LIN {X 0,Y 524.001,Z 123.213,A -85,B 0,C 180,E1 -4868.484,E2 -4868.484} C_VEL
LIN {X 0,Y 524.001,Z 123.208,A -85,B 0,C 180,E1 -4871.74,E2 -4871.74} C_VEL
LIN {X 0,Y 523.991,Z 123.214,A -85,B 0,C 180,E1 -4875.052,E2 -4875.052} C_VEL
LIN {X 0,Y 523.962,Z 123.215,A -85,B 0,C 180,E1 -4877.969,E2 -4877.969} C_VEL
LIN {X 0,Y 523.97,Z 123.219,A -85,B 0,C 180,E1 -4880.41,E2 -4880.41} C_VEL
LIN {X 0,Y 523.909,Z 123.226,A -85,B 0,C 180,E1 -4882.893,E2 -4882.893} C_VEL
LIN {X 0,Y 523.95,Z 123.217,A -85,B 0,C 180,E1 -4885.419,E2 -4885.419} C_VEL
LIN {X 0,Y 523.968,Z 123.218,A -85,B 0,C 180,E1 -4887.999,E2 -4887.999} C_VEL
LIN {X 0,Y 523.945,Z 123.22,A -85,B 0,C 180,E1 -4890.855,E2 -4890.855} C_VEL
LIN {X 0,Y 523.961,Z 123.218,A -85,B 0,C 180,E1 -4893.735,E2 -4893.735} C_VEL
LIN {X 0,Y 524.017,Z 123.347,A -85,B 0,C 180,E1 -4894.881,E2 -4894.881} C_VEL
LIN {X 0,Y 524.386,Z 128.549,A -85,B 0,C 180,E1 -4895.898,E2 -4895.898} C_VEL
LIN {X 0,Y 524.291,Z 138.967,A -85,B 0,C 180,E1 -4897.913,E2 -4897.913} C_VEL
LIN {X 0,Y 525.934,Z 147.356,A -85,B 0,C 180,E1 -4898.081,E2 -4898.081} C_VEL
LIN {X 0,Y 525.786,Z 195.44,A -85,B 0,C 180,E1 -4898.751,E2 -4898.751} C_VEL
LIN {X 0,Y 525.168,Z 201.285,A -85,B 0,C 180,E1 -4898.816,E2 -4898.816} C_VEL
LIN {X 0,Y 519.401,Z 220.267,A -85,B 0,C 180,E1 -4898.921,E2 -4898.921} C_VEL
LIN {X 0,Y 518.753,Z 226.114,A -85,B 0,C 180,E1 -4898.986,E2 -4898.986} C_VEL
LIN {X 0,Y 518.635,Z 247.138,A -85,B 0,C 180,E1 -4899.309,E2 -4899.309} C_VEL
LIN {X 0,Y 518.446,Z 260.421,A -85,B 0,C 180,E1 -4899.672,E2 -4899.672} C_VEL
LIN {X 0,Y 518.242,Z 272.646,A -85,B 0,C 180,E1 -4900.166,E2 -4900.166} C_VEL
LIN {X 0,Y 517.974,Z 284.77,A -85,B 0,C 180,E1 -4900.83,E2 -4900.83} C_VEL
LIN {X 0,Y 517.696,Z 296.092,A -85,B 0,C 180,E1 -4901.626,E2 -4901.626} C_VEL
LIN {X 0,Y 517.426,Z 306.152,A -85,B 0,C 180,E1 -4902.511,E2 -4902.511} C_VEL
LIN {X 0,Y 517.15,Z 314.732,A -85,B 0,C 180,E1 -4903.435,E2 -4903.435} C_VEL
LIN {X 0,Y 516.882,Z 322.531,A -85,B 0,C 180,E1 -4904.452,E2 -4904.452} C_VEL
LIN {X 0,Y 516.675,Z 329.356,A -85,B 0,C 180,E1 -4905.536,E2 -4905.536} C_VEL
LIN {X 0,Y 516.508,Z 336.123,A -85,B 0,C 180,E1 -4906.882,E2 -4906.882} C_VEL
LIN {X 0,Y 516.419,Z 341.098,A -85,B 0,C 180,E1 -4908.176,E2 -4908.176} C_VEL
LIN {X 0,Y 516.322,Z 345.19,A -85,B 0,C 180,E1 -4909.663,E2 -4909.663} C_VEL
LIN {X 0,Y 516.228,Z 347.859,A -85,B 0,C 180,E1 -4911.226,E2 -4911.226} C_VEL
LIN {X 0,Y 516.202,Z 348.684,A -85,B 0,C 180,E1 -4912.218,E2 -4912.218} C_VEL
LIN {X 0,Y 516.215,Z 348.842,A -85,B 0,C 180,E1 -4913.442,E2 -4913.442} C_VEL
LIN {X 0,Y 516.204,Z 347.924,A -85,B 0,C 180,E1 -4914.774,E2 -4914.774} C_VEL
LIN {X 0,Y 516.335,Z 345.799,A -85,B 0,C 180,E1 -4916.128,E2 -4916.128} C_VEL
LIN {X 0,Y 516.364,Z 342.184,A -85,B 0,C 180,E1 -4917.549,E2 -4917.549} C_VEL
LIN {X 0,Y 516.476,Z 337.486,A -85,B 0,C 180,E1 -4918.863,E2 -4918.863} C_VEL
LIN {X 0,Y 516.65,Z 331.294,A -85,B 0,C 180,E1 -4920.186,E2 -4920.186} C_VEL
LIN {X 0,Y 516.858,Z 324.311,A -85,B 0,C 180,E1 -4921.36,E2 -4921.36} C_VEL
LIN {X 0,Y 517.048,Z 316.091,A -85,B 0,C 180,E1 -4922.475,E2 -4922.475} C_VEL
LIN {X 0,Y 517.361,Z 307.081,A -85,B 0,C 180,E1 -4923.47,E2 -4923.47} C_VEL
LIN {X 0,Y 517.635,Z 297.279,A -85,B 0,C 180,E1 -4924.357,E2 -4924.357} C_VEL
LIN {X 0,Y 517.885,Z 286.81,A -85,B 0,C 180,E1 -4925.122,E2 -4925.122} C_VEL
LIN {X 0,Y 518.158,Z 274.714,A -85,B 0,C 180,E1 -4925.813,E2 -4925.813} C_VEL
LIN {X 0,Y 518.398,Z 262.998,A -85,B 0,C 180,E1 -4926.32,E2 -4926.32} C_VEL
LIN {X 0,Y 518.596,Z 250.647,A -85,B 0,C 180,E1 -4926.7,E2 -4926.7} C_VEL
LIN {X 0,Y 518.693,Z 236.856,A -85,B 0,C 180,E1 -4926.953,E2 -4926.953} C_VEL
LIN {X 0,Y 519.143,Z 148.357,A -85,B 0,C 180,E1 -4928.196,E2 -4928.196} C_VEL
LIN {X 0,Y 517.213,Z 138.968,A -85,B 0,C 180,E1 -4928.398,E2 -4928.398} C_VEL
LIN {X 0,Y 517.29,Z 127.147,A -85,B 0,C 180,E1 -4930.764,E2 -4930.764} C_VEL
LIN {X 0,Y 516.945,Z 124.095,A -85,B 0,C 180,E1 -4931.42,E2 -4931.42} C_VEL
LIN {X 0,Y 516.945,Z 124.089,A -85,B 0,C 180,E1 -4934.854,E2 -4934.854} C_VEL
LIN {X 0,Y 516.966,Z 124.086,A -85,B 0,C 180,E1 -4938.234,E2 -4938.234} C_VEL
LIN {X 0,Y 516.965,Z 124.091,A -85,B 0,C 180,E1 -4941.4,E2 -4941.4} C_VEL
LIN {X 0,Y 517.003,Z 124.085,A -85,B 0,C 180,E1 -4943.757,E2 -4943.757} C_VEL
LIN {X 0,Y 517.009,Z 124.081,A -85,B 0,C 180,E1 -4946.883,E2 -4946.883} C_VEL
LIN {X 0,Y 517.093,Z 124.075,A -85,B 0,C 180,E1 -4949.221,E2 -4949.221} C_VEL
LIN {X 0,Y 517.084,Z 124.07,A -85,B 0,C 180,E1 -4952.337,E2 -4952.337} C_VEL
LIN {X 0,Y 517.027,Z 124.082,A -85,B 0,C 180,E1 -4955.46,E2 -4955.46} C_VEL
LIN {X 0,Y 516.956,Z 124.088,A -85,B 0,C 180,E1 -4958.601,E2 -4958.601} C_VEL
LIN {X 0,Y 516.952,Z 124.087,A -85,B 0,C 180,E1 -4961.807,E2 -4961.807} C_VEL
LIN {X 0,Y 516.945,Z 124.093,A -85,B 0,C 180,E1 -4965.146,E2 -4965.146} C_VEL
LIN {X 0,Y 516.916,Z 124.092,A -85,B 0,C 180,E1 -4968.222,E2 -4968.222} C_VEL
LIN {X 0,Y 516.912,Z 124.098,A -85,B 0,C 180,E1 -4970.701,E2 -4970.701} C_VEL
LIN {X 0,Y 516.903,Z 124.093,A -85,B 0,C 180,E1 -4974.072,E2 -4974.072} C_VEL
LIN {X 0,Y 516.924,Z 124.099,A -85,B 0,C 180,E1 -4976.658,E2 -4976.658} C_VEL
LIN {X 0,Y 516.909,Z 124.092,A -85,B 0,C 180,E1 -4979.523,E2 -4979.523} C_VEL
LIN {X 0,Y 516.893,Z 124.103,A -85,B 0,C 180,E1 -4982.543,E2 -4982.543} C_VEL
LIN {X 0,Y 516.865,Z 124.097,A -85,B 0,C 180,E1 -4985.329,E2 -4985.329} C_VEL
LIN {X 0,Y 516.88,Z 124.098,A -85,B 0,C 180,E1 -4987.943,E2 -4987.943} C_VEL
LIN {X 0,Y 516.882,Z 124.098,A -85,B 0,C 180,E1 -4990.741,E2 -4990.741} C_VEL
LIN {X 0,Y 516.883,Z 124.097,A -85,B 0,C 180,E1 -4992.831,E2 -4992.831} C_VEL
LIN {X 0,Y 516.921,Z 124.09,A -85,B 0,C 180,E1 -4995.01,E2 -4995.01} C_VEL
LIN {X 0,Y 516.913,Z 124.096,A -85,B 0,C 180,E1 -4998.398,E2 -4998.398} C_VEL
LIN {X 0,Y 516.881,Z 124.095,A -85,B 0,C 180,E1 -5001.284,E2 -5001.284} C_VEL
LIN {X 0,Y 516.885,Z 124.1,A -85,B 0,C 180,E1 -5004.221,E2 -5004.221} C_VEL
LIN {X 0,Y 516.893,Z 124.094,A -85,B 0,C 180,E1 -5007.053,E2 -5007.053} C_VEL
LIN {X 0,Y 516.899,Z 124.101,A -85,B 0,C 180,E1 -5009.797,E2 -5009.797} C_VEL
LIN {X 0,Y 516.924,Z 124.091,A -85,B 0,C 180,E1 -5012.467,E2 -5012.467} C_VEL
LIN {X 0,Y 516.873,Z 124.097,A -85,B 0,C 180,E1 -5015.07,E2 -5015.07} C_VEL
LIN {X 0,Y 516.866,Z 124.105,A -85,B 0,C 180,E1 -5017.622,E2 -5017.622} C_VEL
LIN {X 0,Y 516.93,Z 124.091,A -85,B 0,C 180,E1 -5020.13,E2 -5020.13} C_VEL
LIN {X 0,Y 516.927,Z 124.089,A -85,B 0,C 180,E1 -5022.596,E2 -5022.596} C_VEL
LIN {X 0,Y 516.949,Z 124.089,A -85,B 0,C 180,E1 -5025.03,E2 -5025.03} C_VEL
LIN {X 0,Y 516.964,Z 124.085,A -85,B 0,C 180,E1 -5028.234,E2 -5028.234} C_VEL
LIN {X 0,Y 516.968,Z 124.092,A -85,B 0,C 180,E1 -5031.4,E2 -5031.4} C_VEL
LIN {X 0,Y 517.014,Z 124.081,A -85,B 0,C 180,E1 -5033.757,E2 -5033.757} C_VEL
LIN {X 0,Y 517.084,Z 124.072,A -85,B 0,C 180,E1 -5037.663,E2 -5037.663} C_VEL
LIN {X 0,Y 517.091,Z 124.073,A -85,B 0,C 180,E1 -5040.779,E2 -5040.779} C_VEL
LIN {X 0,Y 517.011,Z 124.086,A -85,B 0,C 180,E1 -5043.117,E2 -5043.117} C_VEL
LIN {X 0,Y 517.002,Z 124.081,A -85,B 0,C 180,E1 -5046.243,E2 -5046.243} C_VEL
LIN {X 0,Y 516.951,Z 124.088,A -85,B 0,C 180,E1 -5049.389,E2 -5049.389} C_VEL
LIN {X 0,Y 516.951,Z 124.086,A -85,B 0,C 180,E1 -5051.807,E2 -5051.807} C_VEL
LIN {X 0,Y 516.943,Z 124.09,A -85,B 0,C 180,E1 -5055.147,E2 -5055.147} C_VEL
LIN {X 0,Y 516.924,Z 124.093,A -85,B 0,C 180,E1 -5058.222,E2 -5058.222} C_VEL
LIN {X 0,Y 516.912,Z 124.098,A -85,B 0,C 180,E1 -5060.702,E2 -5060.702} C_VEL
LIN {X 0,Y 516.903,Z 124.095,A -85,B 0,C 180,E1 -5064.073,E2 -5064.073} C_VEL
LIN {X 0,Y 516.924,Z 124.095,A -85,B 0,C 180,E1 -5066.658,E2 -5066.658} C_VEL
LIN {X 0,Y 516.911,Z 124.092,A -85,B 0,C 180,E1 -5069.524,E2 -5069.524} C_VEL
LIN {X 0,Y 516.895,Z 124.098,A -85,B 0,C 180,E1 -5072.544,E2 -5072.544} C_VEL
LIN {X 0,Y 516.866,Z 124.097,A -85,B 0,C 180,E1 -5075.33,E2 -5075.33} C_VEL
LIN {X 0,Y 516.882,Z 124.101,A -85,B 0,C 180,E1 -5077.944,E2 -5077.944} C_VEL
LIN {X 0,Y 516.905,Z 124.093,A -85,B 0,C 180,E1 -5080.74,E2 -5080.74} C_VEL
LIN {X 0,Y 516.883,Z 124.102,A -85,B 0,C 180,E1 -5083.903,E2 -5083.903} C_VEL
LIN {X 0,Y 516.883,Z 124.101,A -85,B 0,C 180,E1 -5086.107,E2 -5086.107} C_VEL
LIN {X 0,Y 516.906,Z 124.093,A -85,B 0,C 180,E1 -5089.261,E2 -5089.261} C_VEL
LIN {X 0,Y 516.865,Z 124.1,A -85,B 0,C 180,E1 -5092.275,E2 -5092.275} C_VEL
LIN {X 0,Y 516.884,Z 124.096,A -85,B 0,C 180,E1 -5095.176,E2 -5095.176} C_VEL
LIN {X 0,Y 516.875,Z 124.1,A -85,B 0,C 180,E1 -5097.975,E2 -5097.975} C_VEL
LIN {X 0,Y 516.924,Z 124.092,A -85,B 0,C 180,E1 -5100.696,E2 -5100.696} C_VEL
LIN {X 0,Y 516.945,Z 124.096,A -85,B 0,C 180,E1 -5103.804,E2 -5103.804} C_VEL
LIN {X 0,Y 516.98,Z 124.198,A -85,B 0,C 180,E1 -5104.457,E2 -5104.457} C_VEL
LIN {X 0,Y 518.589,Z 132.719,A -85,B 0,C 180,E1 -5105.837,E2 -5105.837} C_VEL
LIN {X 0,Y 518.195,Z 147.747,A -85,B 0,C 180,E1 -5108.101,E2 -5108.101} C_VEL
LIN {X 0,Y 517.814,Z 164.388,A -85,B 0,C 180,E1 -5110.578,E2 -5110.578} C_VEL
LIN {X 0,Y 517.443,Z 183.777,A -85,B 0,C 180,E1 -5113.428,E2 -5113.428} C_VEL
LIN {X 0,Y 517.219,Z 191.987,A -85,B 0,C 180,E1 -5114.624,E2 -5114.624} C_VEL
LIN {X 0,Y 518.995,Z 205.511,A -85,B 0,C 180,E1 -5114.873,E2 -5114.873} C_VEL
LIN {X 0,Y 518.582,Z 300.996,A -85,B 0,C 180,E1 -5116.231,E2 -5116.231} C_VEL
LIN {X 0,Y 518.283,Z 314.183,A -85,B 0,C 180,E1 -5116.572,E2 -5116.572} C_VEL
LIN {X 0,Y 518.026,Z 326.893,A -85,B 0,C 180,E1 -5117.065,E2 -5117.065} C_VEL
LIN {X 0,Y 517.759,Z 338.435,A -85,B 0,C 180,E1 -5117.67,E2 -5117.67} C_VEL
LIN {X 0,Y 517.447,Z 349.9,A -85,B 0,C 180,E1 -5118.443,E2 -5118.443} C_VEL
LIN {X 0,Y 517.156,Z 360.428,A -85,B 0,C 180,E1 -5119.33,E2 -5119.33} C_VEL
LIN {X 0,Y 516.86,Z 369.035,A -85,B 0,C 180,E1 -5120.214,E2 -5120.214} C_VEL
LIN {X 0,Y 516.674,Z 376.981,A -85,B 0,C 180,E1 -5121.198,E2 -5121.198} C_VEL
LIN {X 0,Y 516.515,Z 384.746,A -85,B 0,C 180,E1 -5122.376,E2 -5122.376} C_VEL
LIN {X 0,Y 516.374,Z 391.895,A -85,B 0,C 180,E1 -5123.749,E2 -5123.749} C_VEL
LIN {X 0,Y 516.312,Z 396.653,A -85,B 0,C 180,E1 -5124.924,E2 -5124.924} C_VEL
LIN {X 0,Y 516.37,Z 400.293,A -85,B 0,C 180,E1 -5126.098,E2 -5126.098} C_VEL
LIN {X 0,Y 516.327,Z 402.167,A -85,B 0,C 180,E1 -5126.879,E2 -5126.879} C_VEL
LIN {X 0,Y 516.266,Z 403.569,A -85,B 0,C 180,E1 -5127.659,E2 -5127.659} C_VEL
LIN {X 0,Y 516.182,Z 405.175,A -85,B 0,C 180,E1 -5129.22,E2 -5129.22} C_VEL
LIN {X 0,Y 516.186,Z 405.389,A -85,B 0,C 180,E1 -5130,E2 -5130} C_VEL
LIN {X 0,Y 516.182,Z 405.167,A -85,B 0,C 180,E1 -5130.78,E2 -5130.78} C_VEL
LIN {X 0,Y 516.266,Z 403.546,A -85,B 0,C 180,E1 -5132.341,E2 -5132.341} C_VEL
LIN {X 0,Y 516.327,Z 402.135,A -85,B 0,C 180,E1 -5133.121,E2 -5133.121} C_VEL
LIN {X 0,Y 516.312,Z 399.164,A -85,B 0,C 180,E1 -5134.293,E2 -5134.293} C_VEL
LIN {X 0,Y 516.388,Z 395.149,A -85,B 0,C 180,E1 -5135.467,E2 -5135.467} C_VEL
LIN {X 0,Y 516.427,Z 388.964,A -85,B 0,C 180,E1 -5136.84,E2 -5136.84} C_VEL
LIN {X 0,Y 516.564,Z 382.225,A -85,B 0,C 180,E1 -5138.016,E2 -5138.016} C_VEL
LIN {X 0,Y 516.751,Z 373.857,A -85,B 0,C 180,E1 -5139.195,E2 -5139.195} C_VEL
LIN {X 0,Y 516.952,Z 365.274,A -85,B 0,C 180,E1 -5140.18,E2 -5140.18} C_VEL
LIN {X 0,Y 517.294,Z 354.681,A -85,B 0,C 180,E1 -5141.163,E2 -5141.163} C_VEL
LIN {X 0,Y 517.565,Z 343.007,A -85,B 0,C 180,E1 -5142.033,E2 -5142.033} C_VEL
LIN {X 0,Y 517.91,Z 330.721,A -85,B 0,C 180,E1 -5142.739,E2 -5142.739} C_VEL
LIN {X 0,Y 518.17,Z 318.202,A -85,B 0,C 180,E1 -5143.281,E2 -5143.281} C_VEL
LIN {X 0,Y 518.48,Z 305.218,A -85,B 0,C 180,E1 -5143.672,E2 -5143.672} C_VEL
LIN {X 0,Y 518.647,Z 289.599,A -85,B 0,C 180,E1 -5143.942,E2 -5143.942} C_VEL
LIN {X 0,Y 518.951,Z 204.029,A -85,B 0,C 180,E1 -5145.145,E2 -5145.145} C_VEL
LIN {X 0,Y 517.226,Z 191.497,A -85,B 0,C 180,E1 -5145.39,E2 -5145.39} C_VEL
LIN {X 0,Y 517.649,Z 169.331,A -85,B 0,C 180,E1 -5148.606,E2 -5148.606} C_VEL
LIN {X 0,Y 518.082,Z 149.697,A -85,B 0,C 180,E1 -5151.485,E2 -5151.485} C_VEL
LIN {X 0,Y 518.414,Z 132.799,A -85,B 0,C 180,E1 -5153.998,E2 -5153.998} C_VEL
LIN {X 0,Y 516.945,Z 124.094,A -85,B 0,C 180,E1 -5155.383,E2 -5155.383} C_VEL
LIN {X 0,Y 516.92,Z 124.1,A -85,B 0,C 180,E1 -5158.415,E2 -5158.415} C_VEL
LIN {X 0,Y 516.89,Z 124.096,A -85,B 0,C 180,E1 -5161.109,E2 -5161.109} C_VEL
LIN {X 0,Y 516.909,Z 124.098,A -85,B 0,C 180,E1 -5163.966,E2 -5163.966} C_VEL
LIN {X 0,Y 516.877,Z 124.1,A -85,B 0,C 180,E1 -5166.746,E2 -5166.746} C_VEL
LIN {X 0,Y 516.904,Z 124.097,A -85,B 0,C 180,E1 -5169.719,E2 -5169.719} C_VEL
LIN {X 0,Y 516.919,Z 124.096,A -85,B 0,C 180,E1 -5171.774,E2 -5171.774} C_VEL
LIN {X 0,Y 516.923,Z 124.092,A -85,B 0,C 180,E1 -5175.01,E2 -5175.01} C_VEL
LIN {X 0,Y 516.923,Z 124.094,A -85,B 0,C 180,E1 -5178.397,E2 -5178.397} C_VEL
LIN {X 0,Y 516.886,Z 124.095,A -85,B 0,C 180,E1 -5181.284,E2 -5181.284} C_VEL
LIN {X 0,Y 516.87,Z 124.101,A -85,B 0,C 180,E1 -5184.219,E2 -5184.219} C_VEL
LIN {X 0,Y 516.894,Z 124.093,A -85,B 0,C 180,E1 -5187.053,E2 -5187.053} C_VEL
LIN {X 0,Y 516.891,Z 124.1,A -85,B 0,C 180,E1 -5189.796,E2 -5189.796} C_VEL
LIN {X 0,Y 516.925,Z 124.09,A -85,B 0,C 180,E1 -5192.467,E2 -5192.467} C_VEL
LIN {X 0,Y 516.874,Z 124.097,A -85,B 0,C 180,E1 -5195.07,E2 -5195.07} C_VEL
LIN {X 0,Y 516.867,Z 124.102,A -85,B 0,C 180,E1 -5197.621,E2 -5197.621} C_VEL
LIN {X 0,Y 516.931,Z 124.089,A -85,B 0,C 180,E1 -5200.13,E2 -5200.13} C_VEL
LIN {X 0,Y 516.928,Z 124.089,A -85,B 0,C 180,E1 -5202.596,E2 -5202.596} C_VEL
LIN {X 0,Y 516.949,Z 124.089,A -85,B 0,C 180,E1 -5205.03,E2 -5205.03} C_VEL
LIN {X 0,Y 516.964,Z 124.084,A -85,B 0,C 180,E1 -5208.233,E2 -5208.233} C_VEL
LIN {X 0,Y 516.968,Z 124.09,A -85,B 0,C 180,E1 -5211.399,E2 -5211.399} C_VEL
LIN {X 0,Y 517.014,Z 124.081,A -85,B 0,C 180,E1 -5213.757,E2 -5213.757} C_VEL
LIN {X 0,Y 517.084,Z 124.072,A -85,B 0,C 180,E1 -5217.663,E2 -5217.663} C_VEL
LIN {X 0,Y 517.091,Z 124.073,A -85,B 0,C 180,E1 -5220.779,E2 -5220.779} C_VEL
LIN {X 0,Y 517.011,Z 124.086,A -85,B 0,C 180,E1 -5223.117,E2 -5223.117} C_VEL
LIN {X 0,Y 517.001,Z 124.08,A -85,B 0,C 180,E1 -5226.243,E2 -5226.243} C_VEL
LIN {X 0,Y 516.95,Z 124.089,A -85,B 0,C 180,E1 -5229.389,E2 -5229.389} C_VEL
LIN {X 0,Y 516.95,Z 124.087,A -85,B 0,C 180,E1 -5231.807,E2 -5231.807} C_VEL
LIN {X 0,Y 516.942,Z 124.091,A -85,B 0,C 180,E1 -5235.146,E2 -5235.146} C_VEL
LIN {X 0,Y 516.923,Z 124.094,A -85,B 0,C 180,E1 -5238.222,E2 -5238.222} C_VEL
LIN {X 0,Y 516.91,Z 124.1,A -85,B 0,C 180,E1 -5240.701,E2 -5240.701} C_VEL
LIN {X 0,Y 516.901,Z 124.099,A -85,B 0,C 180,E1 -5244.072,E2 -5244.072} C_VEL
LIN {X 0,Y 516.924,Z 124.099,A -85,B 0,C 180,E1 -5246.658,E2 -5246.658} C_VEL
LIN {X 0,Y 516.909,Z 124.094,A -85,B 0,C 180,E1 -5249.524,E2 -5249.524} C_VEL
LIN {X 0,Y 516.899,Z 124.102,A -85,B 0,C 180,E1 -5252.544,E2 -5252.544} C_VEL
LIN {X 0,Y 517.005,Z 124.223,A -85,B 0,C 180,E1 -5254.757,E2 -5254.757} C_VEL
LIN {X 0,Y 517.418,Z 129.161,A -85,B 0,C 180,E1 -5255.737,E2 -5255.737} C_VEL
LIN {X 0,Y 517.292,Z 139.212,A -85,B 0,C 180,E1 -5257.689,E2 -5257.689} C_VEL
LIN {X 0,Y 519.145,Z 148.956,A -85,B 0,C 180,E1 -5257.898,E2 -5257.898} C_VEL
LIN {X 0,Y 518.753,Z 226.114,A -85,B 0,C 180,E1 -5258.986,E2 -5258.986} C_VEL
LIN {X 0,Y 518.13,Z 231.958,A -85,B 0,C 180,E1 -5259.048,E2 -5259.048} C_VEL
LIN {X 0,Y 512.865,Z 248.977,A -85,B 0,C 180,E1 -5259.187,E2 -5259.187} C_VEL
LIN {X 0,Y 511.745,Z 254.689,A -85,B 0,C 180,E1 -5259.302,E2 -5259.302} C_VEL
LIN {X 0,Y 511.611,Z 256.599,A -85,B 0,C 180,E1 -5259.354,E2 -5259.354} C_VEL
LIN {X 0,Y 511.364,Z 269.736,A -85,B 0,C 180,E1 -5259.842,E2 -5259.842} C_VEL
LIN {X 0,Y 511.144,Z 282.069,A -85,B 0,C 180,E1 -5260.474,E2 -5260.474} C_VEL
LIN {X 0,Y 510.88,Z 292.825,A -85,B 0,C 180,E1 -5261.188,E2 -5261.188} C_VEL
LIN {X 0,Y 510.5,Z 304.216,A -85,B 0,C 180,E1 -5262.146,E2 -5262.146} C_VEL
LIN {X 0,Y 510.164,Z 313.422,A -85,B 0,C 180,E1 -5263.104,E2 -5263.104} C_VEL
LIN {X 0,Y 509.887,Z 322.109,A -85,B 0,C 180,E1 -5264.215,E2 -5264.215} C_VEL
LIN {X 0,Y 509.676,Z 329.071,A -85,B 0,C 180,E1 -5265.312,E2 -5265.312} C_VEL
LIN {X 0,Y 509.533,Z 334.709,A -85,B 0,C 180,E1 -5266.398,E2 -5266.398} C_VEL
LIN {X 0,Y 509.36,Z 340.58,A -85,B 0,C 180,E1 -5267.846,E2 -5267.846} C_VEL
LIN {X 0,Y 509.284,Z 344.042,A -85,B 0,C 180,E1 -5268.981,E2 -5268.981} C_VEL
LIN {X 0,Y 509.267,Z 345.461,A -85,B 0,C 180,E1 -5269.563,E2 -5269.563} C_VEL
LIN {X 0,Y 509.175,Z 347.461,A -85,B 0,C 180,E1 -5270.62,E2 -5270.62} C_VEL
LIN {X 0,Y 509.118,Z 348.887,A -85,B 0,C 180,E1 -5271.891,E2 -5271.891} C_VEL
LIN {X 0,Y 509.116,Z 349.284,A -85,B 0,C 180,E1 -5273.192,E2 -5273.192} C_VEL
LIN {X 0,Y 509.127,Z 348.543,A -85,B 0,C 180,E1 -5274.566,E2 -5274.566} C_VEL
LIN {X 0,Y 509.217,Z 346.672,A -85,B 0,C 180,E1 -5275.903,E2 -5275.903} C_VEL
LIN {X 0,Y 509.28,Z 343.088,A -85,B 0,C 180,E1 -5277.439,E2 -5277.439} C_VEL
LIN {X 0,Y 509.403,Z 338.431,A -85,B 0,C 180,E1 -5278.802,E2 -5278.802} C_VEL
LIN {X 0,Y 509.604,Z 331.923,A -85,B 0,C 180,E1 -5280.233,E2 -5280.233} C_VEL
LIN {X 0,Y 509.813,Z 325.436,A -85,B 0,C 180,E1 -5281.357,E2 -5281.357} C_VEL
LIN {X 0,Y 510.045,Z 317.213,A -85,B 0,C 180,E1 -5282.51,E2 -5282.51} C_VEL
LIN {X 0,Y 510.341,Z 308.303,A -85,B 0,C 180,E1 -5283.524,E2 -5283.524} C_VEL
LIN {X 0,Y 510.697,Z 297.412,A -85,B 0,C 180,E1 -5284.53,E2 -5284.53} C_VEL
LIN {X 0,Y 511.02,Z 285.851,A -85,B 0,C 180,E1 -5285.368,E2 -5285.368} C_VEL
LIN {X 0,Y 511.263,Z 274.343,A -85,B 0,C 180,E1 -5286.023,E2 -5286.023} C_VEL
LIN {X 0,Y 511.536,Z 262.797,A -85,B 0,C 180,E1 -5286.52,E2 -5286.52} C_VEL
LIN {X 0,Y 511.717,Z 250.546,A -85,B 0,C 180,E1 -5286.895,E2 -5286.895} C_VEL
LIN {X 0,Y 511.848,Z 234.68,A -85,B 0,C 180,E1 -5287.175,E2 -5287.175} C_VEL
LIN {X 0,Y 512.315,Z 149.359,A -85,B 0,C 180,E1 -5288.393,E2 -5288.393} C_VEL
LIN {X 0,Y 510.206,Z 139.259,A -85,B 0,C 180,E1 -5288.617,E2 -5288.617} C_VEL
LIN {X 0,Y 510.286,Z 127.887,A -85,B 0,C 180,E1 -5290.907,E2 -5290.907} C_VEL
LIN {X 0,Y 509.884,Z 124.975,A -85,B 0,C 180,E1 -5291.517,E2 -5291.517} C_VEL
LIN {X 0,Y 509.911,Z 124.965,A -85,B 0,C 180,E1 -5294.819,E2 -5294.819} C_VEL
LIN {X 0,Y 509.901,Z 124.967,A -85,B 0,C 180,E1 -5298.124,E2 -5298.124} C_VEL
LIN {X 0,Y 509.911,Z 124.968,A -85,B 0,C 180,E1 -5301.28,E2 -5301.28} C_VEL
LIN {X 0,Y 509.954,Z 124.964,A -85,B 0,C 180,E1 -5303.67,E2 -5303.67} C_VEL
LIN {X 0,Y 509.951,Z 124.96,A -85,B 0,C 180,E1 -5306.84,E2 -5306.84} C_VEL
LIN {X 0,Y 510.063,Z 124.951,A -85,B 0,C 180,E1 -5309.211,E2 -5309.211} C_VEL
LIN {X 0,Y 510.055,Z 124.945,A -85,B 0,C 180,E1 -5312.369,E2 -5312.369} C_VEL
LIN {X 0,Y 509.978,Z 124.959,A -85,B 0,C 180,E1 -5315.536,E2 -5315.536} C_VEL
LIN {X 0,Y 509.904,Z 124.967,A -85,B 0,C 180,E1 -5318.72,E2 -5318.72} C_VEL
LIN {X 0,Y 509.905,Z 124.964,A -85,B 0,C 180,E1 -5321.932,E2 -5321.932} C_VEL
LIN {X 0,Y 509.894,Z 124.97,A -85,B 0,C 180,E1 -5325.242,E2 -5325.242} C_VEL
LIN {X 0,Y 509.861,Z 124.973,A -85,B 0,C 180,E1 -5328.484,E2 -5328.484} C_VEL
LIN {X 0,Y 509.85,Z 124.977,A -85,B 0,C 180,E1 -5331.002,E2 -5331.002} C_VEL
LIN {X 0,Y 509.864,Z 124.974,A -85,B 0,C 180,E1 -5334.426,E2 -5334.426} C_VEL
LIN {X 0,Y 509.883,Z 124.97,A -85,B 0,C 180,E1 -5337.056,E2 -5337.056} C_VEL
LIN {X 0,Y 509.856,Z 124.97,A -85,B 0,C 180,E1 -5339.751,E2 -5339.751} C_VEL
LIN {X 0,Y 509.866,Z 124.974,A -85,B 0,C 180,E1 -5342.773,E2 -5342.773} C_VEL
LIN {X 0,Y 509.825,Z 124.974,A -85,B 0,C 180,E1 -5345.578,E2 -5345.578} C_VEL
LIN {X 0,Y 509.849,Z 124.979,A -85,B 0,C 180,E1 -5348.338,E2 -5348.338} C_VEL
LIN {X 0,Y 509.855,Z 124.97,A -85,B 0,C 180,E1 -5351.425,E2 -5351.425} C_VEL
LIN {X 0,Y 509.855,Z 124.973,A -85,B 0,C 180,E1 -5354.668,E2 -5354.668} C_VEL
LIN {X 0,Y 509.855,Z 124.979,A -85,B 0,C 180,E1 -5358.103,E2 -5358.103} C_VEL
LIN {X 0,Y 509.846,Z 124.973,A -85,B 0,C 180,E1 -5360.648,E2 -5360.648} C_VEL
LIN {X 0,Y 509.831,Z 124.977,A -85,B 0,C 180,E1 -5363.648,E2 -5363.648} C_VEL
LIN {X 0,Y 509.859,Z 124.971,A -85,B 0,C 180,E1 -5366.539,E2 -5366.539} C_VEL
LIN {X 0,Y 509.848,Z 124.973,A -85,B 0,C 180,E1 -5369.335,E2 -5369.335} C_VEL
LIN {X 0,Y 509.89,Z 124.971,A -85,B 0,C 180,E1 -5372.054,E2 -5372.054} C_VEL
LIN {X 0,Y 509.838,Z 124.972,A -85,B 0,C 180,E1 -5374.702,E2 -5374.702} C_VEL
LIN {X 0,Y 509.824,Z 124.98,A -85,B 0,C 180,E1 -5377.458,E2 -5377.458} C_VEL
LIN {X 0,Y 509.915,Z 124.968,A -85,B 0,C 180,E1 -5379.845,E2 -5379.845} C_VEL
LIN {X 0,Y 509.883,Z 124.971,A -85,B 0,C 180,E1 -5383.175,E2 -5383.175} C_VEL
LIN {X 0,Y 509.871,Z 124.974,A -85,B 0,C 180,E1 -5385.634,E2 -5385.634} C_VEL
LIN {X 0,Y 509.912,Z 124.965,A -85,B 0,C 180,E1 -5388.875,E2 -5388.875} C_VEL
LIN {X 0,Y 509.95,Z 124.959,A -85,B 0,C 180,E1 -5392.079,E2 -5392.079} C_VEL
LIN {X 0,Y 509.984,Z 124.955,A -85,B 0,C 180,E1 -5394.464,E2 -5394.464} C_VEL
LIN {X 0,Y 510.055,Z 124.948,A -85,B 0,C 180,E1 -5397.631,E2 -5397.631} C_VEL
LIN {X 0,Y 510.062,Z 124.949,A -85,B 0,C 180,E1 -5400.79,E2 -5400.79} C_VEL
LIN {X 0,Y 509.954,Z 124.965,A -85,B 0,C 180,E1 -5403.16,E2 -5403.16} C_VEL
LIN {X 0,Y 509.953,Z 124.959,A -85,B 0,C 180,E1 -5406.33,E2 -5406.33} C_VEL
LIN {X 0,Y 509.914,Z 124.969,A -85,B 0,C 180,E1 -5408.72,E2 -5408.72} C_VEL
LIN {X 0,Y 509.903,Z 124.964,A -85,B 0,C 180,E1 -5411.932,E2 -5411.932} C_VEL
LIN {X 0,Y 509.893,Z 124.968,A -85,B 0,C 180,E1 -5415.242,E2 -5415.242} C_VEL
LIN {X 0,Y 509.888,Z 124.967,A -85,B 0,C 180,E1 -5418.001,E2 -5418.001} C_VEL
LIN {X 0,Y 509.849,Z 124.974,A -85,B 0,C 180,E1 -5421.002,E2 -5421.002} C_VEL
LIN {X 0,Y 509.864,Z 124.977,A -85,B 0,C 180,E1 -5424.426,E2 -5424.426} C_VEL
LIN {X 0,Y 509.883,Z 124.968,A -85,B 0,C 180,E1 -5427.056,E2 -5427.056} C_VEL
LIN {X 0,Y 509.857,Z 124.971,A -85,B 0,C 180,E1 -5429.751,E2 -5429.751} C_VEL
LIN {X 0,Y 509.873,Z 124.97,A -85,B 0,C 180,E1 -5432.774,E2 -5432.774} C_VEL
LIN {X 0,Y 509.825,Z 124.975,A -85,B 0,C 180,E1 -5435.579,E2 -5435.579} C_VEL
LIN {X 0,Y 509.852,Z 124.977,A -85,B 0,C 180,E1 -5438.338,E2 -5438.338} C_VEL
LIN {X 0,Y 509.866,Z 124.97,A -85,B 0,C 180,E1 -5441.425,E2 -5441.425} C_VEL
LIN {X 0,Y 509.858,Z 124.971,A -85,B 0,C 180,E1 -5444.668,E2 -5444.668} C_VEL
LIN {X 0,Y 509.863,Z 124.975,A -85,B 0,C 180,E1 -5448.103,E2 -5448.103} C_VEL
LIN {X 0,Y 509.861,Z 124.97,A -85,B 0,C 180,E1 -5450.649,E2 -5450.649} C_VEL
LIN {X 0,Y 509.826,Z 124.981,A -85,B 0,C 180,E1 -5453.647,E2 -5453.647} C_VEL
LIN {X 0,Y 509.86,Z 124.97,A -85,B 0,C 180,E1 -5456.539,E2 -5456.539} C_VEL
LIN {X 0,Y 509.847,Z 124.976,A -85,B 0,C 180,E1 -5459.335,E2 -5459.335} C_VEL
LIN {X 0,Y 509.894,Z 124.971,A -85,B 0,C 180,E1 -5462.055,E2 -5462.055} C_VEL
LIN {X 0,Y 509.922,Z 125.039,A -85,B 0,C 180,E1 -5464.269,E2 -5464.269} C_VEL
LIN {X 0,Y 511.562,Z 133.486,A -85,B 0,C 180,E1 -5465.66,E2 -5465.66} C_VEL
LIN {X 0,Y 511.402,Z 144.615,A -85,B 0,C 180,E1 -5467.369,E2 -5467.369} C_VEL
LIN {X 0,Y 510.907,Z 161.255,A -85,B 0,C 180,E1 -5469.886,E2 -5469.886} C_VEL
LIN {X 0,Y 510.559,Z 177.872,A -85,B 0,C 180,E1 -5472.372,E2 -5472.372} C_VEL
LIN {X 0,Y 510.222,Z 191.609,A -85,B 0,C 180,E1 -5474.406,E2 -5474.406} C_VEL
LIN {X 0,Y 512.161,Z 206.457,A -85,B 0,C 180,E1 -5474.685,E2 -5474.685} C_VEL
LIN {X 0,Y 511.681,Z 300.479,A -85,B 0,C 180,E1 -5476.041,E2 -5476.041} C_VEL
LIN {X 0,Y 511.374,Z 313.709,A -85,B 0,C 180,E1 -5476.387,E2 -5476.387} C_VEL
LIN {X 0,Y 511.097,Z 326.443,A -85,B 0,C 180,E1 -5476.886,E2 -5476.886} C_VEL
LIN {X 0,Y 510.783,Z 338.439,A -85,B 0,C 180,E1 -5477.526,E2 -5477.526} C_VEL
LIN {X 0,Y 510.446,Z 349.479,A -85,B 0,C 180,E1 -5478.283,E2 -5478.283} C_VEL
LIN {X 0,Y 510.14,Z 360.015,A -85,B 0,C 180,E1 -5479.181,E2 -5479.181} C_VEL
LIN {X 0,Y 509.819,Z 368.628,A -85,B 0,C 180,E1 -5480.078,E2 -5480.078} C_VEL
LIN {X 0,Y 509.626,Z 376.58,A -85,B 0,C 180,E1 -5481.075,E2 -5481.075} C_VEL
LIN {X 0,Y 509.427,Z 384.35,A -85,B 0,C 180,E1 -5482.27,E2 -5482.27} C_VEL
LIN {X 0,Y 509.309,Z 390.68,A -85,B 0,C 180,E1 -5483.483,E2 -5483.483} C_VEL
LIN {X 0,Y 509.241,Z 396.264,A -85,B 0,C 180,E1 -5484.853,E2 -5484.853} C_VEL
LIN {X 0,Y 509.275,Z 399.905,A -85,B 0,C 180,E1 -5486.043,E2 -5486.043} C_VEL
LIN {X 0,Y 509.241,Z 401.78,A -85,B 0,C 180,E1 -5486.835,E2 -5486.835} C_VEL
LIN {X 0,Y 509.196,Z 403.184,A -85,B 0,C 180,E1 -5487.627,E2 -5487.627} C_VEL
LIN {X 0,Y 509.094,Z 404.788,A -85,B 0,C 180,E1 -5489.209,E2 -5489.209} C_VEL
LIN {X 0,Y 509.097,Z 405.002,A -85,B 0,C 180,E1 -5490,E2 -5490} C_VEL
LIN {X 0,Y 509.094,Z 404.779,A -85,B 0,C 180,E1 -5490.791,E2 -5490.791} C_VEL
LIN {X 0,Y 509.196,Z 403.154,A -85,B 0,C 180,E1 -5492.373,E2 -5492.373} C_VEL
LIN {X 0,Y 509.241,Z 401.74,A -85,B 0,C 180,E1 -5493.164,E2 -5493.164} C_VEL
LIN {X 0,Y 509.205,Z 398.763,A -85,B 0,C 180,E1 -5494.353,E2 -5494.353} C_VEL
LIN {X 0,Y 509.294,Z 394.744,A -85,B 0,C 180,E1 -5495.543,E2 -5495.543} C_VEL
LIN {X 0,Y 509.343,Z 388.66,A -85,B 0,C 180,E1 -5496.914,E2 -5496.914} C_VEL
LIN {X 0,Y 509.483,Z 381.803,A -85,B 0,C 180,E1 -5498.128,E2 -5498.128} C_VEL
LIN {X 0,Y 509.702,Z 373.43,A -85,B 0,C 180,E1 -5499.324,E2 -5499.324} C_VEL
LIN {X 0,Y 509.931,Z 364.836,A -85,B 0,C 180,E1 -5500.321,E2 -5500.321} C_VEL
LIN {X 0,Y 510.298,Z 354.232,A -85,B 0,C 180,E1 -5501.318,E2 -5501.318} C_VEL
LIN {X 0,Y 510.565,Z 343.307,A -85,B 0,C 180,E1 -5502.147,E2 -5502.147} C_VEL
LIN {X 0,Y 510.896,Z 332.214,A -85,B 0,C 180,E1 -5502.816,E2 -5502.816} C_VEL
LIN {X 0,Y 511.181,Z 320.308,A -85,B 0,C 180,E1 -5503.365,E2 -5503.365} C_VEL
LIN {X 0,Y 511.538,Z 306.59,A -85,B 0,C 180,E1 -5503.811,E2 -5503.811} C_VEL
LIN {X 0,Y 511.733,Z 294.27,A -85,B 0,C 180,E1 -5504.059,E2 -5504.059} C_VEL
LIN {X 0,Y 512.026,Z 204.679,A -85,B 0,C 180,E1 -5505.339,E2 -5505.339} C_VEL
LIN {X 0,Y 510.192,Z 191.082,A -85,B 0,C 180,E1 -5505.607,E2 -5505.607} C_VEL
LIN {X 0,Y 510.688,Z 168.909,A -85,B 0,C 180,E1 -5508.869,E2 -5508.869} C_VEL
LIN {X 0,Y 511.077,Z 149.267,A -85,B 0,C 180,E1 -5511.795,E2 -5511.795} C_VEL
LIN {X 0,Y 511.485,Z 135.208,A -85,B 0,C 180,E1 -5513.912,E2 -5513.912} C_VEL
LIN {X 0,Y 510.858,Z 129.761,A -85,B 0,C 180,E1 -5514.772,E2 -5514.772} C_VEL
LIN {X 0,Y 509.921,Z 124.97,A -85,B 0,C 180,E1 -5515.567,E2 -5515.567} C_VEL
LIN {X 0,Y 509.878,Z 124.974,A -85,B 0,C 180,E1 -5518.844,E2 -5518.844} C_VEL
LIN {X 0,Y 509.821,Z 124.977,A -85,B 0,C 180,E1 -5521.59,E2 -5521.59} C_VEL
LIN {X 0,Y 509.848,Z 124.981,A -85,B 0,C 180,E1 -5524.413,E2 -5524.413} C_VEL
LIN {X 0,Y 509.818,Z 124.978,A -85,B 0,C 180,E1 -5527.34,E2 -5527.34} C_VEL
LIN {X 0,Y 509.863,Z 124.977,A -85,B 0,C 180,E1 -5530.38,E2 -5530.38} C_VEL
LIN {X 0,Y 509.824,Z 124.976,A -85,B 0,C 180,E1 -5533.062,E2 -5533.062} C_VEL
LIN {X 0,Y 509.831,Z 124.981,A -85,B 0,C 180,E1 -5535.792,E2 -5535.792} C_VEL
LIN {X 0,Y 509.866,Z 124.971,A -85,B 0,C 180,E1 -5538.575,E2 -5538.575} C_VEL
LIN {X 0,Y 509.852,Z 124.977,A -85,B 0,C 180,E1 -5541.786,E2 -5541.786} C_VEL
LIN {X 0,Y 509.829,Z 124.974,A -85,B 0,C 180,E1 -5544.622,E2 -5544.622} C_VEL
LIN {X 0,Y 509.86,Z 124.973,A -85,B 0,C 180,E1 -5547.481,E2 -5547.481} C_VEL
LIN {X 0,Y 509.857,Z 124.97,A -85,B 0,C 180,E1 -5550.273,E2 -5550.273} C_VEL
LIN {X 0,Y 509.882,Z 124.968,A -85,B 0,C 180,E1 -5552.944,E2 -5552.944} C_VEL
LIN {X 0,Y 509.85,Z 124.978,A -85,B 0,C 180,E1 -5555.573,E2 -5555.573} C_VEL
LIN {X 0,Y 509.82,Z 124.975,A -85,B 0,C 180,E1 -5558.148,E2 -5558.148} C_VEL
LIN {X 0,Y 509.863,Z 124.968,A -85,B 0,C 180,E1 -5560.681,E2 -5560.681} C_VEL
LIN {X 0,Y 509.883,Z 124.971,A -85,B 0,C 180,E1 -5563.174,E2 -5563.174} C_VEL
LIN {X 0,Y 509.872,Z 124.974,A -85,B 0,C 180,E1 -5565.634,E2 -5565.634} C_VEL
LIN {X 0,Y 509.912,Z 124.965,A -85,B 0,C 180,E1 -5568.874,E2 -5568.874} C_VEL
LIN {X 0,Y 509.95,Z 124.957,A -85,B 0,C 180,E1 -5572.078,E2 -5572.078} C_VEL
LIN {X 0,Y 509.984,Z 124.956,A -85,B 0,C 180,E1 -5574.464,E2 -5574.464} C_VEL
LIN {X 0,Y 510.054,Z 124.948,A -85,B 0,C 180,E1 -5577.631,E2 -5577.631} C_VEL
LIN {X 0,Y 510.061,Z 124.949,A -85,B 0,C 180,E1 -5580.789,E2 -5580.789} C_VEL
LIN {X 0,Y 509.953,Z 124.965,A -85,B 0,C 180,E1 -5583.16,E2 -5583.16} C_VEL
LIN {X 0,Y 509.952,Z 124.959,A -85,B 0,C 180,E1 -5586.33,E2 -5586.33} C_VEL
LIN {X 0,Y 509.913,Z 124.971,A -85,B 0,C 180,E1 -5588.72,E2 -5588.72} C_VEL
LIN {X 0,Y 509.902,Z 124.965,A -85,B 0,C 180,E1 -5591.932,E2 -5591.932} C_VEL
LIN {X 0,Y 509.891,Z 124.969,A -85,B 0,C 180,E1 -5595.242,E2 -5595.242} C_VEL
LIN {X 0,Y 509.886,Z 124.968,A -85,B 0,C 180,E1 -5598.001,E2 -5598.001} C_VEL
LIN {X 0,Y 509.848,Z 124.975,A -85,B 0,C 180,E1 -5601.002,E2 -5601.002} C_VEL
LIN {X 0,Y 509.862,Z 124.98,A -85,B 0,C 180,E1 -5604.426,E2 -5604.426} C_VEL
LIN {X 0,Y 509.884,Z 124.971,A -85,B 0,C 180,E1 -5607.056,E2 -5607.056} C_VEL
LIN {X 0,Y 509.855,Z 124.974,A -85,B 0,C 180,E1 -5609.751,E2 -5609.751} C_VEL
LIN {X 0,Y 509.875,Z 124.974,A -85,B 0,C 180,E1 -5612.775,E2 -5612.775} C_VEL
LIN {X 0,Y 509.941,Z 125.072,A -85,B 0,C 180,E1 -5614.616,E2 -5614.616} C_VEL
LIN {X 0,Y 510.432,Z 128.617,A -85,B 0,C 180,E1 -5615.33,E2 -5615.33} C_VEL
LIN {X 0,Y 510.316,Z 139.618,A -85,B 0,C 180,E1 -5617.484,E2 -5617.484} C_VEL
LIN {X 0,Y 512.313,Z 149.986,A -85,B 0,C 180,E1 -5617.7,E2 -5617.7} C_VEL
LIN {X 0,Y 511.762,Z 246.544,A -85,B 0,C 180,E1 -5619.102,E2 -5619.102} C_VEL
LIN {X 0,Y 511.611,Z 256.599,A -85,B 0,C 180,E1 -5619.354,E2 -5619.354} C_VEL
LIN {X 0,Y 510.822,Z 262.281,A -85,B 0,C 180,E1 -5619.518,E2 -5619.518} C_VEL
LIN {X 0,Y 507.883,Z 271.4,A -85,B 0,C 180,E1 -5619.81,E2 -5619.81} C_VEL
LIN {X 0,Y 504.938,Z 280.226,A -85,B 0,C 180,E1 -5620.189,E2 -5620.189} C_VEL
LIN {X 0,Y 504.139,Z 285.44,A -85,B 0,C 180,E1 -5620.487,E2 -5620.487} C_VEL
LIN {X 0,Y 503.808,Z 296.866,A -85,B 0,C 180,E1 -5621.311,E2 -5621.311} C_VEL
LIN {X 0,Y 503.458,Z 307.527,A -85,B 0,C 180,E1 -5622.282,E2 -5622.282} C_VEL
LIN {X 0,Y 503.086,Z 317.464,A -85,B 0,C 180,E1 -5623.413,E2 -5623.413} C_VEL
LIN {X 0,Y 502.765,Z 325.406,A -85,B 0,C 180,E1 -5624.528,E2 -5624.528} C_VEL
LIN {X 0,Y 502.554,Z 331.823,A -85,B 0,C 180,E1 -5625.635,E2 -5625.635} C_VEL
LIN {X 0,Y 502.405,Z 338.104,A -85,B 0,C 180,E1 -5627.004,E2 -5627.004} C_VEL
LIN {X 0,Y 502.263,Z 342.886,A -85,B 0,C 180,E1 -5628.37,E2 -5628.37} C_VEL
LIN {X 0,Y 502.201,Z 344.858,A -85,B 0,C 180,E1 -5629.086,E2 -5629.086} C_VEL
LIN {X 0,Y 502.102,Z 347.458,A -85,B 0,C 180,E1 -5630.34,E2 -5630.34} C_VEL
LIN {X 0,Y 502.03,Z 349.336,A -85,B 0,C 180,E1 -5631.978,E2 -5631.978} C_VEL
LIN {X 0,Y 502.043,Z 349.69,A -85,B 0,C 180,E1 -5632.991,E2 -5632.991} C_VEL
LIN {X 0,Y 502.032,Z 349.208,A -85,B 0,C 180,E1 -5634.286,E2 -5634.286} C_VEL
LIN {X 0,Y 502.116,Z 347.547,A -85,B 0,C 180,E1 -5635.67,E2 -5635.67} C_VEL
LIN {X 0,Y 502.191,Z 344.513,A -85,B 0,C 180,E1 -5637.106,E2 -5637.106} C_VEL
LIN {X 0,Y 502.33,Z 339.92,A -85,B 0,C 180,E1 -5638.587,E2 -5638.587} C_VEL
LIN {X 0,Y 502.475,Z 335.052,A -85,B 0,C 180,E1 -5639.767,E2 -5639.767} C_VEL
LIN {X 0,Y 502.642,Z 329.065,A -85,B 0,C 180,E1 -5640.93,E2 -5640.93} C_VEL
LIN {X 0,Y 502.906,Z 321.711,A -85,B 0,C 180,E1 -5642.086,E2 -5642.086} C_VEL
LIN {X 0,Y 503.205,Z 312.846,A -85,B 0,C 180,E1 -5643.212,E2 -5643.212} C_VEL
LIN {X 0,Y 503.565,Z 302.723,A -85,B 0,C 180,E1 -5644.253,E2 -5644.253} C_VEL
LIN {X 0,Y 503.877,Z 292,A -85,B 0,C 180,E1 -5645.138,E2 -5645.138} C_VEL
LIN {X 0,Y 504.271,Z 279.52,A -85,B 0,C 180,E1 -5645.943,E2 -5645.943} C_VEL
LIN {X 0,Y 504.529,Z 267.537,A -85,B 0,C 180,E1 -5646.532,E2 -5646.532} C_VEL
LIN {X 0,Y 504.783,Z 254.261,A -85,B 0,C 180,E1 -5646.992,E2 -5646.992} C_VEL
LIN {X 0,Y 504.941,Z 241.804,A -85,B 0,C 180,E1 -5647.266,E2 -5647.266} C_VEL
LIN {X 0,Y 505.473,Z 150.39,A -85,B 0,C 180,E1 -5648.594,E2 -5648.594} C_VEL
LIN {X 0,Y 503.232,Z 139.535,A -85,B 0,C 180,E1 -5648.845,E2 -5648.845} C_VEL
LIN {X 0,Y 503.349,Z 129.654,A -85,B 0,C 180,E1 -5650.846,E2 -5650.846} C_VEL
LIN {X 0,Y 502.838,Z 125.853,A -85,B 0,C 180,E1 -5651.671,E2 -5651.671} C_VEL
LIN {X 0,Y 502.839,Z 125.846,A -85,B 0,C 180,E1 -5654.663,E2 -5654.663} C_VEL
LIN {X 0,Y 502.876,Z 125.843,A -85,B 0,C 180,E1 -5658.039,E2 -5658.039} C_VEL
LIN {X 0,Y 502.869,Z 125.844,A -85,B 0,C 180,E1 -5661.157,E2 -5661.157} C_VEL
LIN {X 0,Y 502.907,Z 125.844,A -85,B 0,C 180,E1 -5663.581,E2 -5663.581} C_VEL
LIN {X 0,Y 502.894,Z 125.839,A -85,B 0,C 180,E1 -5666.796,E2 -5666.796} C_VEL
LIN {X 0,Y 503.034,Z 125.826,A -85,B 0,C 180,E1 -5669.2,E2 -5669.2} C_VEL
LIN {X 0,Y 502.904,Z 125.841,A -85,B 0,C 180,E1 -5671.602,E2 -5671.602} C_VEL
LIN {X 0,Y 502.896,Z 125.845,A -85,B 0,C 180,E1 -5673.205,E2 -5673.205} C_VEL
LIN {X 0,Y 502.892,Z 125.838,A -85,B 0,C 180,E1 -5676.419,E2 -5676.419} C_VEL
LIN {X 0,Y 502.865,Z 125.846,A -85,B 0,C 180,E1 -5678.843,E2 -5678.843} C_VEL
LIN {X 0,Y 502.846,Z 125.843,A -85,B 0,C 180,E1 -5682.102,E2 -5682.102} C_VEL
LIN {X 0,Y 502.849,Z 125.846,A -85,B 0,C 180,E1 -5685.4,E2 -5685.4} C_VEL
LIN {X 0,Y 502.826,Z 125.853,A -85,B 0,C 180,E1 -5688.752,E2 -5688.752} C_VEL
LIN {X 0,Y 502.783,Z 125.854,A -85,B 0,C 180,E1 -5691.311,E2 -5691.311} C_VEL
LIN {X 0,Y 502.785,Z 125.851,A -85,B 0,C 180,E1 -5693.914,E2 -5693.914} C_VEL
LIN {X 0,Y 502.864,Z 125.848,A -85,B 0,C 180,E1 -5696.566,E2 -5696.566} C_VEL
LIN {X 0,Y 502.822,Z 125.847,A -85,B 0,C 180,E1 -5699.288,E2 -5699.288} C_VEL
LIN {X 0,Y 502.781,Z 125.854,A -85,B 0,C 180,E1 -5702.085,E2 -5702.085} C_VEL
LIN {X 0,Y 502.794,Z 125.852,A -85,B 0,C 180,E1 -5704.966,E2 -5704.966} C_VEL
LIN {X 0,Y 502.792,Z 125.853,A -85,B 0,C 180,E1 -5707.954,E2 -5707.954} C_VEL
LIN {X 0,Y 502.819,Z 125.847,A -85,B 0,C 180,E1 -5711.066,E2 -5711.066} C_VEL
LIN {X 0,Y 502.8,Z 125.854,A -85,B 0,C 180,E1 -5714.532,E2 -5714.532} C_VEL
LIN {X 0,Y 502.794,Z 125.854,A -85,B 0,C 180,E1 -5717.861,E2 -5717.861} C_VEL
LIN {X 0,Y 502.801,Z 125.849,A -85,B 0,C 180,E1 -5721.024,E2 -5721.024} C_VEL
LIN {X 0,Y 502.781,Z 125.858,A -85,B 0,C 180,E1 -5724.168,E2 -5724.168} C_VEL
LIN {X 0,Y 502.83,Z 125.845,A -85,B 0,C 180,E1 -5726.993,E2 -5726.993} C_VEL
LIN {X 0,Y 502.815,Z 125.853,A -85,B 0,C 180,E1 -5730.065,E2 -5730.065} C_VEL
LIN {X 0,Y 502.83,Z 125.846,A -85,B 0,C 180,E1 -5732.533,E2 -5732.533} C_VEL
LIN {X 0,Y 502.801,Z 125.852,A -85,B 0,C 180,E1 -5735.305,E2 -5735.305} C_VEL
LIN {X 0,Y 502.778,Z 125.858,A -85,B 0,C 180,E1 -5737.826,E2 -5737.826} C_VEL
LIN {X 0,Y 502.823,Z 125.847,A -85,B 0,C 180,E1 -5740.4,E2 -5740.4} C_VEL
LIN {X 0,Y 502.832,Z 125.847,A -85,B 0,C 180,E1 -5742.932,E2 -5742.932} C_VEL
LIN {X 0,Y 502.85,Z 125.851,A -85,B 0,C 180,E1 -5745.429,E2 -5745.429} C_VEL
LIN {X 0,Y 502.876,Z 125.841,A -85,B 0,C 180,E1 -5748.717,E2 -5748.717} C_VEL
LIN {X 0,Y 502.9,Z 125.838,A -85,B 0,C 180,E1 -5751.967,E2 -5751.967} C_VEL
LIN {X 0,Y 502.94,Z 125.832,A -85,B 0,C 180,E1 -5754.387,E2 -5754.387} C_VEL
LIN {X 0,Y 503.024,Z 125.824,A -85,B 0,C 180,E1 -5757.598,E2 -5757.598} C_VEL
LIN {X 0,Y 503.026,Z 125.821,A -85,B 0,C 180,E1 -5760,E2 -5760} C_VEL
LIN {X 0,Y 503.024,Z 125.822,A -85,B 0,C 180,E1 -5762.402,E2 -5762.402} C_VEL
LIN {X 0,Y 502.932,Z 125.834,A -85,B 0,C 180,E1 -5765.614,E2 -5765.614} C_VEL
LIN {X 0,Y 502.9,Z 125.837,A -85,B 0,C 180,E1 -5768.034,E2 -5768.034} C_VEL
LIN {X 0,Y 502.876,Z 125.842,A -85,B 0,C 180,E1 -5771.283,E2 -5771.283} C_VEL
LIN {X 0,Y 502.844,Z 125.85,A -85,B 0,C 180,E1 -5774.571,E2 -5774.571} C_VEL
LIN {X 0,Y 502.861,Z 125.842,A -85,B 0,C 180,E1 -5777.907,E2 -5777.907} C_VEL
LIN {X 0,Y 502.828,Z 125.854,A -85,B 0,C 180,E1 -5780.536,E2 -5780.536} C_VEL
LIN {X 0,Y 502.79,Z 125.852,A -85,B 0,C 180,E1 -5783.041,E2 -5783.041} C_VEL
LIN {X 0,Y 502.839,Z 125.845,A -85,B 0,C 180,E1 -5785.676,E2 -5785.676} C_VEL
LIN {X 0,Y 502.839,Z 125.853,A -85,B 0,C 180,E1 -5788.373,E2 -5788.373} C_VEL
LIN {X 0,Y 502.792,Z 125.85,A -85,B 0,C 180,E1 -5791.499,E2 -5791.499} C_VEL
LIN {X 0,Y 502.803,Z 125.854,A -85,B 0,C 180,E1 -5793.994,E2 -5793.994} C_VEL
LIN {X 0,Y 502.778,Z 125.852,A -85,B 0,C 180,E1 -5797.178,E2 -5797.178} C_VEL
LIN {X 0,Y 502.822,Z 125.854,A -85,B 0,C 180,E1 -5800.012,E2 -5800.012} C_VEL
LIN {X 0,Y 502.774,Z 125.853,A -85,B 0,C 180,E1 -5803.231,E2 -5803.231} C_VEL
LIN {X 0,Y 502.791,Z 125.855,A -85,B 0,C 180,E1 -5805.662,E2 -5805.662} C_VEL
LIN {X 0,Y 502.828,Z 125.846,A -85,B 0,C 180,E1 -5809.004,E2 -5809.004} C_VEL
LIN {X 0,Y 502.795,Z 125.855,A -85,B 0,C 180,E1 -5812.047,E2 -5812.047} C_VEL
LIN {X 0,Y 502.8,Z 125.85,A -85,B 0,C 180,E1 -5815.035,E2 -5815.035} C_VEL
LIN {X 0,Y 502.785,Z 125.856,A -85,B 0,C 180,E1 -5817.916,E2 -5817.916} C_VEL
LIN {X 0,Y 502.826,Z 125.849,A -85,B 0,C 180,E1 -5820.713,E2 -5820.713} C_VEL
LIN {X 0,Y 502.867,Z 125.849,A -85,B 0,C 180,E1 -5823.992,E2 -5823.992} C_VEL
LIN {X 0,Y 502.905,Z 126.061,A -85,B 0,C 180,E1 -5824.106,E2 -5824.106} C_VEL
LIN {X 0,Y 504.732,Z 135.91,A -85,B 0,C 180,E1 -5825.747,E2 -5825.747} C_VEL
LIN {X 0,Y 504.254,Z 152.573,A -85,B 0,C 180,E1 -5828.325,E2 -5828.325} C_VEL
LIN {X 0,Y 503.688,Z 173.986,A -85,B 0,C 180,E1 -5831.589,E2 -5831.589} C_VEL
LIN {X 0,Y 503.21,Z 191.544,A -85,B 0,C 180,E1 -5834.195,E2 -5834.195} C_VEL
LIN {X 0,Y 505.297,Z 206.941,A -85,B 0,C 180,E1 -5834.487,E2 -5834.487} C_VEL
LIN {X 0,Y 504.786,Z 299.931,A -85,B 0,C 180,E1 -5835.847,E2 -5835.847} C_VEL
LIN {X 0,Y 504.457,Z 313.217,A -85,B 0,C 180,E1 -5836.197,E2 -5836.197} C_VEL
LIN {X 0,Y 504.141,Z 325.981,A -85,B 0,C 180,E1 -5836.702,E2 -5836.702} C_VEL
LIN {X 0,Y 503.819,Z 337.264,A -85,B 0,C 180,E1 -5837.304,E2 -5837.304} C_VEL
LIN {X 0,Y 503.404,Z 349.053,A -85,B 0,C 180,E1 -5838.116,E2 -5838.116} C_VEL
LIN {X 0,Y 503.126,Z 359.602,A -85,B 0,C 180,E1 -5839.028,E2 -5839.028} C_VEL
LIN {X 0,Y 502.791,Z 368.222,A -85,B 0,C 180,E1 -5839.937,E2 -5839.937} C_VEL
LIN {X 0,Y 502.561,Z 376.178,A -85,B 0,C 180,E1 -5840.948,E2 -5840.948} C_VEL
LIN {X 0,Y 502.363,Z 383.954,A -85,B 0,C 180,E1 -5842.16,E2 -5842.16} C_VEL
LIN {X 0,Y 502.216,Z 391.11,A -85,B 0,C 180,E1 -5843.572,E2 -5843.572} C_VEL
LIN {X 0,Y 502.17,Z 395.875,A -85,B 0,C 180,E1 -5844.781,E2 -5844.781} C_VEL
LIN {X 0,Y 502.165,Z 399.516,A -85,B 0,C 180,E1 -5845.987,E2 -5845.987} C_VEL
LIN {X 0,Y 502.158,Z 401.394,A -85,B 0,C 180,E1 -5846.791,E2 -5846.791} C_VEL
LIN {X 0,Y 502.128,Z 402.799,A -85,B 0,C 180,E1 -5847.593,E2 -5847.593} C_VEL
LIN {X 0,Y 502.009,Z 404.401,A -85,B 0,C 180,E1 -5849.198,E2 -5849.198} C_VEL
LIN {X 0,Y 502.01,Z 404.614,A -85,B 0,C 180,E1 -5850,E2 -5850} C_VEL
LIN {X 0,Y 502.01,Z 404.39,A -85,B 0,C 180,E1 -5850.802,E2 -5850.802} C_VEL
LIN {X 0,Y 502.128,Z 402.762,A -85,B 0,C 180,E1 -5852.406,E2 -5852.406} C_VEL
LIN {X 0,Y 502.158,Z 401.345,A -85,B 0,C 180,E1 -5853.209,E2 -5853.209} C_VEL
LIN {X 0,Y 502.104,Z 398.363,A -85,B 0,C 180,E1 -5854.415,E2 -5854.415} C_VEL
LIN {X 0,Y 502.201,Z 394.338,A -85,B 0,C 180,E1 -5855.622,E2 -5855.622} C_VEL
LIN {X 0,Y 502.281,Z 388.247,A -85,B 0,C 180,E1 -5857.012,E2 -5857.012} C_VEL
LIN {X 0,Y 502.42,Z 381.383,A -85,B 0,C 180,E1 -5858.243,E2 -5858.243} C_VEL
LIN {X 0,Y 502.652,Z 373.002,A -85,B 0,C 180,E1 -5859.456,E2 -5859.456} C_VEL
LIN {X 0,Y 502.922,Z 364.402,A -85,B 0,C 180,E1 -5860.467,E2 -5860.467} C_VEL
LIN {X 0,Y 503.273,Z 353.786,A -85,B 0,C 180,E1 -5861.478,E2 -5861.478} C_VEL
LIN {X 0,Y 503.613,Z 342.423,A -85,B 0,C 180,E1 -5862.348,E2 -5862.348} C_VEL
LIN {X 0,Y 503.932,Z 331.748,A -85,B 0,C 180,E1 -5862.996,E2 -5862.996} C_VEL
LIN {X 0,Y 504.247,Z 319.821,A -85,B 0,C 180,E1 -5863.552,E2 -5863.552} C_VEL
LIN {X 0,Y 504.65,Z 306.078,A -85,B 0,C 180,E1 -5864.003,E2 -5864.003} C_VEL
LIN {X 0,Y 504.853,Z 293.684,A -85,B 0,C 180,E1 -5864.254,E2 -5864.254} C_VEL
LIN {X 0,Y 505.153,Z 205.316,A -85,B 0,C 180,E1 -5865.538,E2 -5865.538} C_VEL
LIN {X 0,Y 503.192,Z 190.739,A -85,B 0,C 180,E1 -5865.819,E2 -5865.819} C_VEL
LIN {X 0,Y 503.734,Z 168.486,A -85,B 0,C 180,E1 -5869.139,E2 -5869.139} C_VEL
LIN {X 0,Y 504.126,Z 150.269,A -85,B 0,C 180,E1 -5871.896,E2 -5871.896} C_VEL
LIN {X 0,Y 504.553,Z 136.206,A -85,B 0,C 180,E1 -5874.043,E2 -5874.043} C_VEL
LIN {X 0,Y 503.826,Z 130.593,A -85,B 0,C 180,E1 -5874.946,E2 -5874.946} C_VEL
LIN {X 0,Y 502.877,Z 125.847,A -85,B 0,C 180,E1 -5875.757,E2 -5875.757} C_VEL
LIN {X 0,Y 502.842,Z 125.853,A -85,B 0,C 180,E1 -5878.372,E2 -5878.372} C_VEL
LIN {X 0,Y 502.794,Z 125.852,A -85,B 0,C 180,E1 -5881.498,E2 -5881.498} C_VEL
LIN {X 0,Y 502.805,Z 125.855,A -85,B 0,C 180,E1 -5883.994,E2 -5883.994} C_VEL
LIN {X 0,Y 502.779,Z 125.855,A -85,B 0,C 180,E1 -5887.177,E2 -5887.177} C_VEL
LIN {X 0,Y 502.823,Z 125.855,A -85,B 0,C 180,E1 -5890.011,E2 -5890.011} C_VEL
LIN {X 0,Y 502.774,Z 125.855,A -85,B 0,C 180,E1 -5893.231,E2 -5893.231} C_VEL
LIN {X 0,Y 502.79,Z 125.856,A -85,B 0,C 180,E1 -5895.661,E2 -5895.661} C_VEL
LIN {X 0,Y 502.827,Z 125.847,A -85,B 0,C 180,E1 -5899.004,E2 -5899.004} C_VEL
LIN {X 0,Y 502.794,Z 125.858,A -85,B 0,C 180,E1 -5902.046,E2 -5902.046} C_VEL
LIN {X 0,Y 502.798,Z 125.85,A -85,B 0,C 180,E1 -5905.034,E2 -5905.034} C_VEL
LIN {X 0,Y 502.782,Z 125.859,A -85,B 0,C 180,E1 -5907.915,E2 -5907.915} C_VEL
LIN {X 0,Y 502.823,Z 125.845,A -85,B 0,C 180,E1 -5910.712,E2 -5910.712} C_VEL
LIN {X 0,Y 502.861,Z 125.847,A -85,B 0,C 180,E1 -5913.439,E2 -5913.439} C_VEL
LIN {X 0,Y 502.774,Z 125.854,A -85,B 0,C 180,E1 -5916.085,E2 -5916.085} C_VEL
LIN {X 0,Y 502.782,Z 125.851,A -85,B 0,C 180,E1 -5918.689,E2 -5918.689} C_VEL
LIN {X 0,Y 502.829,Z 125.849,A -85,B 0,C 180,E1 -5921.248,E2 -5921.248} C_VEL
LIN {X 0,Y 502.821,Z 125.849,A -85,B 0,C 180,E1 -5923.767,E2 -5923.767} C_VEL
LIN {X 0,Y 502.834,Z 125.845,A -85,B 0,C 180,E1 -5926.255,E2 -5926.255} C_VEL
LIN {X 0,Y 502.876,Z 125.84,A -85,B 0,C 180,E1 -5928.717,E2 -5928.717} C_VEL
LIN {X 0,Y 502.9,Z 125.836,A -85,B 0,C 180,E1 -5931.966,E2 -5931.966} C_VEL
LIN {X 0,Y 502.94,Z 125.833,A -85,B 0,C 180,E1 -5934.386,E2 -5934.386} C_VEL
LIN {X 0,Y 503.024,Z 125.824,A -85,B 0,C 180,E1 -5937.598,E2 -5937.598} C_VEL
LIN {X 0,Y 503.026,Z 125.82,A -85,B 0,C 180,E1 -5940,E2 -5940} C_VEL
LIN {X 0,Y 503.024,Z 125.823,A -85,B 0,C 180,E1 -5942.402,E2 -5942.402} C_VEL
LIN {X 0,Y 502.932,Z 125.833,A -85,B 0,C 180,E1 -5945.613,E2 -5945.613} C_VEL
LIN {X 0,Y 502.899,Z 125.838,A -85,B 0,C 180,E1 -5948.033,E2 -5948.033} C_VEL
LIN {X 0,Y 502.875,Z 125.842,A -85,B 0,C 180,E1 -5951.283,E2 -5951.283} C_VEL
LIN {X 0,Y 502.842,Z 125.85,A -85,B 0,C 180,E1 -5954.571,E2 -5954.571} C_VEL
LIN {X 0,Y 502.86,Z 125.843,A -85,B 0,C 180,E1 -5957.907,E2 -5957.907} C_VEL
LIN {X 0,Y 502.826,Z 125.854,A -85,B 0,C 180,E1 -5960.536,E2 -5960.536} C_VEL
LIN {X 0,Y 502.789,Z 125.856,A -85,B 0,C 180,E1 -5963.041,E2 -5963.041} C_VEL
LIN {X 0,Y 502.838,Z 125.848,A -85,B 0,C 180,E1 -5965.676,E2 -5965.676} C_VEL
LIN {X 0,Y 502.838,Z 125.852,A -85,B 0,C 180,E1 -5968.373,E2 -5968.373} C_VEL
LIN {X 0,Y 502.794,Z 125.853,A -85,B 0,C 180,E1 -5971.5,E2 -5971.5} C_VEL
LIN {X 0,Y 502.873,Z 125.872,A -85,B 0,C 180,E1 -5974.456,E2 -5974.456} C_VEL
LIN {X 0,Y 503.466,Z 130.548,A -85,B 0,C 180,E1 -5975.402,E2 -5975.402} C_VEL
LIN {X 0,Y 503.363,Z 139.957,A -85,B 0,C 180,E1 -5977.255,E2 -5977.255} C_VEL
LIN {X 0,Y 505.484,Z 150.53,A -85,B 0,C 180,E1 -5977.488,E2 -5977.488} C_VEL
LIN {X 0,Y 504.879,Z 246.524,A -85,B 0,C 180,E1 -5978.9,E2 -5978.9} C_VEL
LIN {X 0,Y 504.653,Z 260.13,A -85,B 0,C 180,E1 -5979.268,E2 -5979.268} C_VEL
LIN {X 0,Y 504.449,Z 272.874,A -85,B 0,C 180,E1 -5979.785,E2 -5979.785} C_VEL
LIN {X 0,Y 504.188,Z 284.311,A -85,B 0,C 180,E1 -5980.415,E2 -5980.415} C_VEL
LIN {X 0,Y 504.139,Z 285.44,A -85,B 0,C 180,E1 -5980.487,E2 -5980.487} C_VEL
LIN {X 0,Y 503.339,Z 290.572,A -85,B 0,C 180,E1 -5980.813,E2 -5980.813} C_VEL
LIN {X 0,Y 500.351,Z 298.696,A -85,B 0,C 180,E1 -5981.361,E2 -5981.361} C_VEL
LIN {X 0,Y 497.297,Z 306.377,A -85,B 0,C 180,E1 -5981.987,E2 -5981.987} C_VEL
LIN {X 0,Y 496.402,Z 310.759,A -85,B 0,C 180,E1 -5982.431,E2 -5982.431} C_VEL
LIN {X 0,Y 495.993,Z 320.141,A -85,B 0,C 180,E1 -5983.58,E2 -5983.58} C_VEL
LIN {X 0,Y 495.665,Z 328.466,A -85,B 0,C 180,E1 -5984.851,E2 -5984.851} C_VEL
LIN {X 0,Y 495.475,Z 334.371,A -85,B 0,C 180,E1 -5985.97,E2 -5985.97} C_VEL
LIN {X 0,Y 495.318,Z 339.103,A -85,B 0,C 180,E1 -5987.074,E2 -5987.074} C_VEL
LIN {X 0,Y 495.216,Z 342.855,A -85,B 0,C 180,E1 -5988.163,E2 -5988.163} C_VEL
LIN {X 0,Y 495.103,Z 345.748,A -85,B 0,C 180,E1 -5989.234,E2 -5989.234} C_VEL
LIN {X 0,Y 495.042,Z 347.835,A -85,B 0,C 180,E1 -5990.294,E2 -5990.294} C_VEL
LIN {X 0,Y 494.97,Z 349.219,A -85,B 0,C 180,E1 -5991.346,E2 -5991.346} C_VEL
LIN {X 0,Y 494.942,Z 350.021,A -85,B 0,C 180,E1 -5992.672,E2 -5992.672} C_VEL
LIN {X 0,Y 494.938,Z 349.755,A -85,B 0,C 180,E1 -5994.036,E2 -5994.036} C_VEL
LIN {X 0,Y 495.008,Z 348.329,A -85,B 0,C 180,E1 -5995.433,E2 -5995.433} C_VEL
LIN {X 0,Y 495.111,Z 345.613,A -85,B 0,C 180,E1 -5996.876,E2 -5996.876} C_VEL
LIN {X 0,Y 495.25,Z 341.323,A -85,B 0,C 180,E1 -5998.369,E2 -5998.369} C_VEL
LIN {X 0,Y 495.408,Z 336.405,A -85,B 0,C 180,E1 -5999.638,E2 -5999.638} C_VEL
LIN {X 0,Y 495.588,Z 329.972,A -85,B 0,C 180,E1 -6000.942,E2 -6000.942} C_VEL
LIN {X 0,Y 495.865,Z 322.752,A -85,B 0,C 180,E1 -6002.114,E2 -6002.114} C_VEL
LIN {X 0,Y 496.223,Z 313.305,A -85,B 0,C 180,E1 -6003.342,E2 -6003.342} C_VEL
LIN {X 0,Y 496.63,Z 302.858,A -85,B 0,C 180,E1 -6004.43,E2 -6004.43} C_VEL
LIN {X 0,Y 496.979,Z 291.822,A -85,B 0,C 180,E1 -6005.344,E2 -6005.344} C_VEL
LIN {X 0,Y 497.366,Z 279.517,A -85,B 0,C 180,E1 -6006.142,E2 -6006.142} C_VEL
LIN {X 0,Y 497.658,Z 267.328,A -85,B 0,C 180,E1 -6006.741,E2 -6006.741} C_VEL
LIN {X 0,Y 497.909,Z 254.499,A -85,B 0,C 180,E1 -6007.187,E2 -6007.187} C_VEL
LIN {X 0,Y 498.088,Z 241.666,A -85,B 0,C 180,E1 -6007.47,E2 -6007.47} C_VEL
LIN {X 0,Y 498.56,Z 150.955,A -85,B 0,C 180,E1 -6008.809,E2 -6008.809} C_VEL
LIN {X 0,Y 496.282,Z 139.885,A -85,B 0,C 180,E1 -6009.063,E2 -6009.063} C_VEL
LIN {X 0,Y 496.329,Z 130.439,A -85,B 0,C 180,E1 -6010.993,E2 -6010.993} C_VEL
LIN {X 0,Y 495.824,Z 126.727,A -85,B 0,C 180,E1 -6011.783,E2 -6011.783} C_VEL
LIN {X 0,Y 495.79,Z 126.727,A -85,B 0,C 180,E1 -6015.217,E2 -6015.217} C_VEL
LIN {X 0,Y 495.851,Z 126.715,A -85,B 0,C 180,E1 -6018.555,E2 -6018.555} C_VEL
LIN {X 0,Y 495.872,Z 126.717,A -85,B 0,C 180,E1 -6021.852,E2 -6021.852} C_VEL
LIN {X 0,Y 495.89,Z 126.71,A -85,B 0,C 180,E1 -6024.307,E2 -6024.307} C_VEL
LIN {X 0,Y 495.994,Z 126.703,A -85,B 0,C 180,E1 -6027.564,E2 -6027.564} C_VEL
LIN {X 0,Y 495.983,Z 126.7,A -85,B 0,C 180,E1 -6030.812,E2 -6030.812} C_VEL
LIN {X 0,Y 495.993,Z 126.697,A -85,B 0,C 180,E1 -6032.436,E2 -6032.436} C_VEL
LIN {X 0,Y 495.885,Z 126.713,A -85,B 0,C 180,E1 -6035.694,E2 -6035.694} C_VEL
LIN {X 0,Y 495.835,Z 126.723,A -85,B 0,C 180,E1 -6038.97,E2 -6038.97} C_VEL
LIN {X 0,Y 495.829,Z 126.718,A -85,B 0,C 180,E1 -6042.035,E2 -6042.035} C_VEL
LIN {X 0,Y 495.824,Z 126.721,A -85,B 0,C 180,E1 -6045.452,E2 -6045.452} C_VEL
LIN {X 0,Y 495.778,Z 126.725,A -85,B 0,C 180,E1 -6048.237,E2 -6048.237} C_VEL
LIN {X 0,Y 495.774,Z 126.732,A -85,B 0,C 180,E1 -6050.756,E2 -6050.756} C_VEL
LIN {X 0,Y 495.747,Z 126.729,A -85,B 0,C 180,E1 -6053.387,E2 -6053.387} C_VEL
LIN {X 0,Y 495.79,Z 126.724,A -85,B 0,C 180,E1 -6056.068,E2 -6056.068} C_VEL
LIN {X 0,Y 495.771,Z 126.731,A -85,B 0,C 180,E1 -6058.815,E2 -6058.815} C_VEL
LIN {X 0,Y 495.754,Z 126.727,A -85,B 0,C 180,E1 -6061.725,E2 -6061.725} C_VEL
LIN {X 0,Y 495.761,Z 126.732,A -85,B 0,C 180,E1 -6064.693,E2 -6064.693} C_VEL
LIN {X 0,Y 495.728,Z 126.73,A -85,B 0,C 180,E1 -6067.562,E2 -6067.562} C_VEL
LIN {X 0,Y 495.765,Z 126.729,A -85,B 0,C 180,E1 -6070.7,E2 -6070.7} C_VEL
LIN {X 0,Y 495.733,Z 126.735,A -85,B 0,C 180,E1 -6074.001,E2 -6074.001} C_VEL
LIN {X 0,Y 495.724,Z 126.731,A -85,B 0,C 180,E1 -6077.117,E2 -6077.117} C_VEL
LIN {X 0,Y 495.757,Z 126.733,A -85,B 0,C 180,E1 -6079.953,E2 -6079.953} C_VEL
LIN {X 0,Y 495.728,Z 126.732,A -85,B 0,C 180,E1 -6082.553,E2 -6082.553} C_VEL
LIN {X 0,Y 495.781,Z 126.726,A -85,B 0,C 180,E1 -6085.457,E2 -6085.457} C_VEL
LIN {X 0,Y 495.754,Z 126.729,A -85,B 0,C 180,E1 -6088.364,E2 -6088.364} C_VEL
LIN {X 0,Y 495.786,Z 126.727,A -85,B 0,C 180,E1 -6091.507,E2 -6091.507} C_VEL
LIN {X 0,Y 495.779,Z 126.73,A -85,B 0,C 180,E1 -6093.932,E2 -6093.932} C_VEL
LIN {X 0,Y 495.757,Z 126.728,A -85,B 0,C 180,E1 -6097.14,E2 -6097.14} C_VEL
LIN {X 0,Y 495.769,Z 126.727,A -85,B 0,C 180,E1 -6100.11,E2 -6100.11} C_VEL
LIN {X 0,Y 495.785,Z 126.723,A -85,B 0,C 180,E1 -6102.682,E2 -6102.682} C_VEL
LIN {X 0,Y 495.793,Z 126.727,A -85,B 0,C 180,E1 -6105.217,E2 -6105.217} C_VEL
LIN {X 0,Y 495.85,Z 126.715,A -85,B 0,C 180,E1 -6108.555,E2 -6108.555} C_VEL
LIN {X 0,Y 495.872,Z 126.714,A -85,B 0,C 180,E1 -6111.852,E2 -6111.852} C_VEL
LIN {X 0,Y 495.897,Z 126.709,A -85,B 0,C 180,E1 -6114.307,E2 -6114.307} C_VEL
LIN {X 0,Y 495.993,Z 126.7,A -85,B 0,C 180,E1 -6117.564,E2 -6117.564} C_VEL
LIN {X 0,Y 495.997,Z 126.697,A -85,B 0,C 180,E1 -6120,E2 -6120} C_VEL
LIN {X 0,Y 495.993,Z 126.699,A -85,B 0,C 180,E1 -6122.436,E2 -6122.436} C_VEL
LIN {X 0,Y 495.888,Z 126.711,A -85,B 0,C 180,E1 -6125.694,E2 -6125.694} C_VEL
LIN {X 0,Y 495.872,Z 126.713,A -85,B 0,C 180,E1 -6128.148,E2 -6128.148} C_VEL
LIN {X 0,Y 495.851,Z 126.716,A -85,B 0,C 180,E1 -6131.445,E2 -6131.445} C_VEL
LIN {X 0,Y 495.789,Z 126.731,A -85,B 0,C 180,E1 -6134.783,E2 -6134.783} C_VEL
LIN {X 0,Y 495.785,Z 126.724,A -85,B 0,C 180,E1 -6137.319,E2 -6137.319} C_VEL
LIN {X 0,Y 495.777,Z 126.725,A -85,B 0,C 180,E1 -6139.89,E2 -6139.89} C_VEL
LIN {X 0,Y 495.759,Z 126.73,A -85,B 0,C 180,E1 -6142.861,E2 -6142.861} C_VEL
LIN {X 0,Y 495.79,Z 126.726,A -85,B 0,C 180,E1 -6146.068,E2 -6146.068} C_VEL
LIN {X 0,Y 495.771,Z 126.728,A -85,B 0,C 180,E1 -6148.815,E2 -6148.815} C_VEL
LIN {X 0,Y 495.755,Z 126.728,A -85,B 0,C 180,E1 -6151.726,E2 -6151.726} C_VEL
LIN {X 0,Y 495.768,Z 126.728,A -85,B 0,C 180,E1 -6154.694,E2 -6154.694} C_VEL
LIN {X 0,Y 495.73,Z 126.731,A -85,B 0,C 180,E1 -6157.562,E2 -6157.562} C_VEL
LIN {X 0,Y 495.78,Z 126.725,A -85,B 0,C 180,E1 -6160.699,E2 -6160.699} C_VEL
LIN {X 0,Y 495.735,Z 126.738,A -85,B 0,C 180,E1 -6164.001,E2 -6164.001} C_VEL
LIN {X 0,Y 495.727,Z 126.731,A -85,B 0,C 180,E1 -6167.117,E2 -6167.117} C_VEL
LIN {X 0,Y 495.791,Z 126.73,A -85,B 0,C 180,E1 -6169.949,E2 -6169.949} C_VEL
LIN {X 0,Y 495.73,Z 126.73,A -85,B 0,C 180,E1 -6172.553,E2 -6172.553} C_VEL
LIN {X 0,Y 495.779,Z 126.729,A -85,B 0,C 180,E1 -6175.457,E2 -6175.457} C_VEL
LIN {X 0,Y 495.757,Z 126.728,A -85,B 0,C 180,E1 -6178.364,E2 -6178.364} C_VEL
LIN {X 0,Y 495.79,Z 126.73,A -85,B 0,C 180,E1 -6181.507,E2 -6181.507} C_VEL
LIN {X 0,Y 495.843,Z 126.748,A -85,B 0,C 180,E1 -6183.884,E2 -6183.884} C_VEL
LIN {X 0,Y 497.776,Z 136.925,A -85,B 0,C 180,E1 -6185.608,E2 -6185.608} C_VEL
LIN {X 0,Y 497.289,Z 152.193,A -85,B 0,C 180,E1 -6188.006,E2 -6188.006} C_VEL
LIN {X 0,Y 496.84,Z 168.827,A -85,B 0,C 180,E1 -6190.585,E2 -6190.585} C_VEL
LIN {X 0,Y 496.298,Z 188.183,A -85,B 0,C 180,E1 -6193.548,E2 -6193.548} C_VEL
LIN {X 0,Y 496.201,Z 190.943,A -85,B 0,C 180,E1 -6193.964,E2 -6193.964} C_VEL
LIN {X 0,Y 498.436,Z 207.802,A -85,B 0,C 180,E1 -6194.287,E2 -6194.287} C_VEL
LIN {X 0,Y 497.894,Z 300.503,A -85,B 0,C 180,E1 -6195.673,E2 -6195.673} C_VEL
LIN {X 0,Y 497.525,Z 313.469,A -85,B 0,C 180,E1 -6196.027,E2 -6196.027} C_VEL
LIN {X 0,Y 497.21,Z 325.503,A -85,B 0,C 180,E1 -6196.513,E2 -6196.513} C_VEL
LIN {X 0,Y 496.857,Z 336.859,A -85,B 0,C 180,E1 -6197.126,E2 -6197.126} C_VEL
LIN {X 0,Y 496.422,Z 348.618,A -85,B 0,C 180,E1 -6197.947,E2 -6197.947} C_VEL
LIN {X 0,Y 496.067,Z 359.174,A -85,B 0,C 180,E1 -6198.87,E2 -6198.87} C_VEL
LIN {X 0,Y 495.757,Z 367.806,A -85,B 0,C 180,E1 -6199.793,E2 -6199.793} C_VEL
LIN {X 0,Y 495.508,Z 375.77,A -85,B 0,C 180,E1 -6200.818,E2 -6200.818} C_VEL
LIN {X 0,Y 495.308,Z 383.556,A -85,B 0,C 180,E1 -6202.048,E2 -6202.048} C_VEL
LIN {X 0,Y 495.128,Z 390.716,A -85,B 0,C 180,E1 -6203.48,E2 -6203.48} C_VEL
LIN {X 0,Y 495.1,Z 395.486,A -85,B 0,C 180,E1 -6204.706,E2 -6204.706} C_VEL
LIN {X 0,Y 495.056,Z 399.127,A -85,B 0,C 180,E1 -6205.93,E2 -6205.93} C_VEL
LIN {X 0,Y 495.077,Z 401.007,A -85,B 0,C 180,E1 -6206.745,E2 -6206.745} C_VEL
LIN {X 0,Y 495.062,Z 402.414,A -85,B 0,C 180,E1 -6207.559,E2 -6207.559} C_VEL
LIN {X 0,Y 494.928,Z 404.015,A -85,B 0,C 180,E1 -6209.186,E2 -6209.186} C_VEL
LIN {X 0,Y 494.926,Z 404.227,A -85,B 0,C 180,E1 -6210,E2 -6210} C_VEL
LIN {X 0,Y 494.966,Z 403.38,A -85,B 0,C 180,E1 -6211.627,E2 -6211.627} C_VEL
LIN {X 0,Y 495.062,Z 402.371,A -85,B 0,C 180,E1 -6212.441,E2 -6212.441} C_VEL
LIN {X 0,Y 495.077,Z 400.95,A -85,B 0,C 180,E1 -6213.255,E2 -6213.255} C_VEL
LIN {X 0,Y 495.009,Z 397.963,A -85,B 0,C 180,E1 -6214.479,E2 -6214.479} C_VEL
LIN {X 0,Y 495.109,Z 393.934,A -85,B 0,C 180,E1 -6215.702,E2 -6215.702} C_VEL
LIN {X 0,Y 495.236,Z 387.736,A -85,B 0,C 180,E1 -6217.133,E2 -6217.133} C_VEL
LIN {X 0,Y 495.345,Z 380.967,A -85,B 0,C 180,E1 -6218.362,E2 -6218.362} C_VEL
LIN {X 0,Y 495.579,Z 372.578,A -85,B 0,C 180,E1 -6219.592,E2 -6219.592} C_VEL
LIN {X 0,Y 495.906,Z 363.971,A -85,B 0,C 180,E1 -6220.617,E2 -6220.617} C_VEL
LIN {X 0,Y 496.248,Z 353.344,A -85,B 0,C 180,E1 -6221.643,E2 -6221.643} C_VEL
LIN {X 0,Y 496.646,Z 341.536,A -85,B 0,C 180,E1 -6222.556,E2 -6222.556} C_VEL
LIN {X 0,Y 497.041,Z 329.308,A -85,B 0,C 180,E1 -6223.283,E2 -6223.283} C_VEL
LIN {X 0,Y 497.443,Z 316.749,A -85,B 0,C 180,E1 -6223.845,E2 -6223.845} C_VEL
LIN {X 0,Y 497.795,Z 303.627,A -85,B 0,C 180,E1 -6224.252,E2 -6224.252} C_VEL
LIN {X 0,Y 497.997,Z 287.866,A -85,B 0,C 180,E1 -6224.533,E2 -6224.533} C_VEL
LIN {X 0,Y 498.341,Z 206.323,A -85,B 0,C 180,E1 -6225.736,E2 -6225.736} C_VEL
LIN {X 0,Y 496.165,Z 190.364,A -85,B 0,C 180,E1 -6226.048,E2 -6226.048} C_VEL
LIN {X 0,Y 496.75,Z 169.491,A -85,B 0,C 180,E1 -6229.204,E2 -6229.204} C_VEL
LIN {X 0,Y 497.287,Z 148.463,A -85,B 0,C 180,E1 -6232.432,E2 -6232.432} C_VEL
LIN {X 0,Y 497.603,Z 137.203,A -85,B 0,C 180,E1 -6234.179,E2 -6234.179} C_VEL
LIN {X 0,Y 496.517,Z 130.096,A -85,B 0,C 180,E1 -6235.351,E2 -6235.351} C_VEL
LIN {X 0,Y 495.844,Z 126.724,A -85,B 0,C 180,E1 -6235.952,E2 -6235.952} C_VEL
LIN {X 0,Y 495.774,Z 126.732,A -85,B 0,C 180,E1 -6238.814,E2 -6238.814} C_VEL
LIN {X 0,Y 495.756,Z 126.73,A -85,B 0,C 180,E1 -6241.725,E2 -6241.725} C_VEL
LIN {X 0,Y 495.77,Z 126.731,A -85,B 0,C 180,E1 -6244.694,E2 -6244.694} C_VEL
LIN {X 0,Y 495.731,Z 126.734,A -85,B 0,C 180,E1 -6247.561,E2 -6247.561} C_VEL
LIN {X 0,Y 495.781,Z 126.728,A -85,B 0,C 180,E1 -6250.698,E2 -6250.698} C_VEL
LIN {X 0,Y 495.735,Z 126.738,A -85,B 0,C 180,E1 -6254,E2 -6254} C_VEL
LIN {X 0,Y 495.726,Z 126.733,A -85,B 0,C 180,E1 -6257.117,E2 -6257.117} C_VEL
LIN {X 0,Y 495.789,Z 126.731,A -85,B 0,C 180,E1 -6259.948,E2 -6259.948} C_VEL
LIN {X 0,Y 495.728,Z 126.732,A -85,B 0,C 180,E1 -6262.553,E2 -6262.553} C_VEL
LIN {X 0,Y 495.777,Z 126.728,A -85,B 0,C 180,E1 -6265.456,E2 -6265.456} C_VEL
LIN {X 0,Y 495.754,Z 126.729,A -85,B 0,C 180,E1 -6268.363,E2 -6268.363} C_VEL
LIN {X 0,Y 495.786,Z 126.727,A -85,B 0,C 180,E1 -6271.507,E2 -6271.507} C_VEL
LIN {X 0,Y 495.779,Z 126.727,A -85,B 0,C 180,E1 -6273.931,E2 -6273.931} C_VEL
LIN {X 0,Y 495.757,Z 126.728,A -85,B 0,C 180,E1 -6277.139,E2 -6277.139} C_VEL
LIN {X 0,Y 495.776,Z 126.724,A -85,B 0,C 180,E1 -6280.11,E2 -6280.11} C_VEL
LIN {X 0,Y 495.785,Z 126.723,A -85,B 0,C 180,E1 -6282.681,E2 -6282.681} C_VEL
LIN {X 0,Y 495.793,Z 126.726,A -85,B 0,C 180,E1 -6285.217,E2 -6285.217} C_VEL
LIN {X 0,Y 495.85,Z 126.714,A -85,B 0,C 180,E1 -6288.555,E2 -6288.555} C_VEL
LIN {X 0,Y 495.871,Z 126.712,A -85,B 0,C 180,E1 -6291.852,E2 -6291.852} C_VEL
LIN {X 0,Y 495.897,Z 126.71,A -85,B 0,C 180,E1 -6294.306,E2 -6294.306} C_VEL
LIN {X 0,Y 495.992,Z 126.701,A -85,B 0,C 180,E1 -6297.564,E2 -6297.564} C_VEL
LIN {X 0,Y 495.997,Z 126.696,A -85,B 0,C 180,E1 -6300,E2 -6300} C_VEL
LIN {X 0,Y 495.992,Z 126.699,A -85,B 0,C 180,E1 -6302.436,E2 -6302.436} C_VEL
LIN {X 0,Y 495.888,Z 126.71,A -85,B 0,C 180,E1 -6305.693,E2 -6305.693} C_VEL
LIN {X 0,Y 495.871,Z 126.714,A -85,B 0,C 180,E1 -6308.148,E2 -6308.148} C_VEL
LIN {X 0,Y 495.849,Z 126.716,A -85,B 0,C 180,E1 -6311.445,E2 -6311.445} C_VEL
LIN {X 0,Y 495.788,Z 126.732,A -85,B 0,C 180,E1 -6314.783,E2 -6314.783} C_VEL
LIN {X 0,Y 495.784,Z 126.725,A -85,B 0,C 180,E1 -6317.319,E2 -6317.319} C_VEL
LIN {X 0,Y 495.775,Z 126.726,A -85,B 0,C 180,E1 -6319.89,E2 -6319.89} C_VEL
LIN {X 0,Y 495.757,Z 126.735,A -85,B 0,C 180,E1 -6322.861,E2 -6322.861} C_VEL
LIN {X 0,Y 495.788,Z 126.73,A -85,B 0,C 180,E1 -6326.068,E2 -6326.068} C_VEL
LIN {X 0,Y 495.77,Z 126.73,A -85,B 0,C 180,E1 -6328.815,E2 -6328.815} C_VEL
LIN {X 0,Y 495.756,Z 126.731,A -85,B 0,C 180,E1 -6331.726,E2 -6331.726} C_VEL
LIN {X 0,Y 495.82,Z 126.728,A -85,B 0,C 180,E1 -6334.294,E2 -6334.294} C_VEL
LIN {X 0,Y 496.51,Z 131.439,A -85,B 0,C 180,E1 -6335.261,E2 -6335.261} C_VEL
LIN {X 0,Y 496.426,Z 140.312,A -85,B 0,C 180,E1 -6337.022,E2 -6337.022} C_VEL
LIN {X 0,Y 498.679,Z 151.054,A -85,B 0,C 180,E1 -6337.27,E2 -6337.27} C_VEL
LIN {X 0,Y 498.018,Z 247.339,A -85,B 0,C 180,E1 -6338.712,E2 -6338.712} C_VEL
LIN {X 0,Y 497.781,Z 260.872,A -85,B 0,C 180,E1 -6339.087,E2 -6339.087} C_VEL
LIN {X 0,Y 497.555,Z 273.238,A -85,B 0,C 180,E1 -6339.598,E2 -6339.598} C_VEL
LIN {X 0,Y 497.276,Z 284.973,A -85,B 0,C 180,E1 -6340.255,E2 -6340.255} C_VEL
LIN {X 0,Y 496.885,Z 296.991,A -85,B 0,C 180,E1 -6341.125,E2 -6341.125} C_VEL
LIN {X 0,Y 496.459,Z 307.81,A -85,B 0,C 180,E1 -6342.117,E2 -6342.117} C_VEL
LIN {X 0,Y 496.402,Z 310.759,A -85,B 0,C 180,E1 -6342.431,E2 -6342.431} C_VEL
LIN {X 0,Y 495.496,Z 315.029,A -85,B 0,C 180,E1 -6342.901,E2 -6342.901} C_VEL
LIN {X 0,Y 492.381,Z 321.572,A -85,B 0,C 180,E1 -6343.683,E2 -6343.683} C_VEL
LIN {X 0,Y 489.344,Z 327.59,A -85,B 0,C 180,E1 -6344.529,E2 -6344.529} C_VEL
LIN {X 0,Y 488.565,Z 330.874,A -85,B 0,C 180,E1 -6345.095,E2 -6345.095} C_VEL
LIN {X 0,Y 488.336,Z 336.739,A -85,B 0,C 180,E1 -6346.307,E2 -6346.307} C_VEL
LIN {X 0,Y 488.204,Z 341.084,A -85,B 0,C 180,E1 -6347.422,E2 -6347.422} C_VEL
LIN {X 0,Y 488.117,Z 344.503,A -85,B 0,C 180,E1 -6348.524,E2 -6348.524} C_VEL
LIN {X 0,Y 487.975,Z 347.367,A -85,B 0,C 180,E1 -6349.758,E2 -6349.758} C_VEL
LIN {X 0,Y 487.892,Z 349.363,A -85,B 0,C 180,E1 -6351.065,E2 -6351.065} C_VEL
LIN {X 0,Y 487.857,Z 350.36,A -85,B 0,C 180,E1 -6352.403,E2 -6352.403} C_VEL
LIN {X 0,Y 487.845,Z 350.291,A -85,B 0,C 180,E1 -6353.797,E2 -6353.797} C_VEL
LIN {X 0,Y 487.897,Z 349.089,A -85,B 0,C 180,E1 -6355.191,E2 -6355.191} C_VEL
LIN {X 0,Y 488.052,Z 346.219,A -85,B 0,C 180,E1 -6356.825,E2 -6356.825} C_VEL
LIN {X 0,Y 488.152,Z 342.664,A -85,B 0,C 180,E1 -6358.15,E2 -6358.15} C_VEL
LIN {X 0,Y 488.272,Z 338.681,A -85,B 0,C 180,E1 -6359.272,E2 -6359.272} C_VEL
LIN {X 0,Y 488.479,Z 333.333,A -85,B 0,C 180,E1 -6360.477,E2 -6360.477} C_VEL
LIN {X 0,Y 488.741,Z 326.767,A -85,B 0,C 180,E1 -6361.671,E2 -6361.671} C_VEL
LIN {X 0,Y 489.057,Z 318.796,A -85,B 0,C 180,E1 -6362.847,E2 -6362.847} C_VEL
LIN {X 0,Y 489.387,Z 309.931,A -85,B 0,C 180,E1 -6363.909,E2 -6363.909} C_VEL
LIN {X 0,Y 489.789,Z 299.782,A -85,B 0,C 180,E1 -6364.899,E2 -6364.899} C_VEL
LIN {X 0,Y 490.182,Z 288.675,A -85,B 0,C 180,E1 -6365.77,E2 -6365.77} C_VEL
LIN {X 0,Y 490.506,Z 276.858,A -85,B 0,C 180,E1 -6366.49,E2 -6366.49} C_VEL
LIN {X 0,Y 490.84,Z 264.872,A -85,B 0,C 180,E1 -6367.043,E2 -6367.043} C_VEL
LIN {X 0,Y 491.102,Z 251.95,A -85,B 0,C 180,E1 -6367.465,E2 -6367.465} C_VEL
LIN {X 0,Y 491.234,Z 236.936,A -85,B 0,C 180,E1 -6367.748,E2 -6367.748} C_VEL
LIN {X 0,Y 491.811,Z 152.206,A -85,B 0,C 180,E1 -6369.014,E2 -6369.014} C_VEL
LIN {X 0,Y 489.31,Z 140.195,A -85,B 0,C 180,E1 -6369.296,E2 -6369.296} C_VEL
LIN {X 0,Y 489.405,Z 132.115,A -85,B 0,C 180,E1 -6370.954,E2 -6370.954} C_VEL
LIN {X 0,Y 488.772,Z 127.605,A -85,B 0,C 180,E1 -6371.925,E2 -6371.925} C_VEL
LIN {X 0,Y 488.762,Z 127.601,A -85,B 0,C 180,E1 -6375,E2 -6375} C_VEL
LIN {X 0,Y 488.805,Z 127.593,A -85,B 0,C 180,E1 -6378.388,E2 -6378.388} C_VEL
LIN {X 0,Y 488.816,Z 127.597,A -85,B 0,C 180,E1 -6381.734,E2 -6381.734} C_VEL
LIN {X 0,Y 488.848,Z 127.588,A -85,B 0,C 180,E1 -6384.224,E2 -6384.224} C_VEL
LIN {X 0,Y 488.961,Z 127.58,A -85,B 0,C 180,E1 -6387.529,E2 -6387.529} C_VEL
LIN {X 0,Y 488.934,Z 127.579,A -85,B 0,C 180,E1 -6390.824,E2 -6390.824} C_VEL
LIN {X 0,Y 488.961,Z 127.573,A -85,B 0,C 180,E1 -6392.471,E2 -6392.471} C_VEL
LIN {X 0,Y 488.842,Z 127.59,A -85,B 0,C 180,E1 -6395.776,E2 -6395.776} C_VEL
LIN {X 0,Y 488.785,Z 127.595,A -85,B 0,C 180,E1 -6398.267,E2 -6398.267} C_VEL
LIN {X 0,Y 488.806,Z 127.594,A -85,B 0,C 180,E1 -6401.612,E2 -6401.612} C_VEL
LIN {X 0,Y 488.762,Z 127.606,A -85,B 0,C 180,E1 -6405,E2 -6405} C_VEL
LIN {X 0,Y 488.747,Z 127.603,A -85,B 0,C 180,E1 -6408.442,E2 -6408.442} C_VEL
LIN {X 0,Y 488.707,Z 127.61,A -85,B 0,C 180,E1 -6411.071,E2 -6411.071} C_VEL
LIN {X 0,Y 488.688,Z 127.607,A -85,B 0,C 180,E1 -6413.746,E2 -6413.746} C_VEL
LIN {X 0,Y 488.791,Z 127.599,A -85,B 0,C 180,E1 -6416.943,E2 -6416.943} C_VEL
LIN {X 0,Y 488.709,Z 127.61,A -85,B 0,C 180,E1 -6420.363,E2 -6420.363} C_VEL
LIN {X 0,Y 488.728,Z 127.602,A -85,B 0,C 180,E1 -6423.483,E2 -6423.483} C_VEL
LIN {X 0,Y 488.681,Z 127.615,A -85,B 0,C 180,E1 -6426.354,E2 -6426.354} C_VEL
LIN {X 0,Y 488.699,Z 127.606,A -85,B 0,C 180,E1 -6429.254,E2 -6429.254} C_VEL
LIN {X 0,Y 488.706,Z 127.606,A -85,B 0,C 180,E1 -6431.6,E2 -6431.6} C_VEL
LIN {X 0,Y 488.711,Z 127.606,A -85,B 0,C 180,E1 -6434.801,E2 -6434.801} C_VEL
LIN {X 0,Y 488.69,Z 127.608,A -85,B 0,C 180,E1 -6437.474,E2 -6437.474} C_VEL
LIN {X 0,Y 488.731,Z 127.605,A -85,B 0,C 180,E1 -6439.677,E2 -6439.677} C_VEL
LIN {X 0,Y 488.68,Z 127.608,A -85,B 0,C 180,E1 -6442.841,E2 -6442.841} C_VEL
LIN {X 0,Y 488.731,Z 127.609,A -85,B 0,C 180,E1 -6445.887,E2 -6445.887} C_VEL
LIN {X 0,Y 488.691,Z 127.607,A -85,B 0,C 180,E1 -6448.82,E2 -6448.82} C_VEL
LIN {X 0,Y 488.743,Z 127.607,A -85,B 0,C 180,E1 -6451.671,E2 -6451.671} C_VEL
LIN {X 0,Y 488.725,Z 127.603,A -85,B 0,C 180,E1 -6454.443,E2 -6454.443} C_VEL
LIN {X 0,Y 488.719,Z 127.605,A -85,B 0,C 180,E1 -6457.153,E2 -6457.153} C_VEL
LIN {X 0,Y 488.723,Z 127.608,A -85,B 0,C 180,E1 -6459.811,E2 -6459.811} C_VEL
LIN {X 0,Y 488.732,Z 127.602,A -85,B 0,C 180,E1 -6462.424,E2 -6462.424} C_VEL
LIN {X 0,Y 488.763,Z 127.6,A -85,B 0,C 180,E1 -6465,E2 -6465} C_VEL
LIN {X 0,Y 488.804,Z 127.593,A -85,B 0,C 180,E1 -6468.388,E2 -6468.388} C_VEL
LIN {X 0,Y 488.816,Z 127.594,A -85,B 0,C 180,E1 -6471.734,E2 -6471.734} C_VEL
LIN {X 0,Y 488.856,Z 127.586,A -85,B 0,C 180,E1 -6474.224,E2 -6474.224} C_VEL
LIN {X 0,Y 488.96,Z 127.577,A -85,B 0,C 180,E1 -6477.529,E2 -6477.529} C_VEL
LIN {X 0,Y 488.952,Z 127.579,A -85,B 0,C 180,E1 -6480.824,E2 -6480.824} C_VEL
LIN {X 0,Y 488.96,Z 127.575,A -85,B 0,C 180,E1 -6482.472,E2 -6482.472} C_VEL
LIN {X 0,Y 488.847,Z 127.588,A -85,B 0,C 180,E1 -6485.776,E2 -6485.776} C_VEL
LIN {X 0,Y 488.816,Z 127.592,A -85,B 0,C 180,E1 -6488.267,E2 -6488.267} C_VEL
LIN {X 0,Y 488.804,Z 127.593,A -85,B 0,C 180,E1 -6491.613,E2 -6491.613} C_VEL
LIN {X 0,Y 488.761,Z 127.603,A -85,B 0,C 180,E1 -6495.001,E2 -6495.001} C_VEL
LIN {X 0,Y 488.754,Z 127.605,A -85,B 0,C 180,E1 -6498.442,E2 -6498.442} C_VEL
LIN {X 0,Y 488.706,Z 127.607,A -85,B 0,C 180,E1 -6501.071,E2 -6501.071} C_VEL
LIN {X 0,Y 488.688,Z 127.608,A -85,B 0,C 180,E1 -6503.746,E2 -6503.746} C_VEL
LIN {X 0,Y 488.791,Z 127.596,A -85,B 0,C 180,E1 -6506.944,E2 -6506.944} C_VEL
LIN {X 0,Y 488.709,Z 127.613,A -85,B 0,C 180,E1 -6510.363,E2 -6510.363} C_VEL
LIN {X 0,Y 488.734,Z 127.602,A -85,B 0,C 180,E1 -6513.484,E2 -6513.484} C_VEL
LIN {X 0,Y 488.682,Z 127.614,A -85,B 0,C 180,E1 -6516.355,E2 -6516.355} C_VEL
LIN {X 0,Y 488.743,Z 127.6,A -85,B 0,C 180,E1 -6519.251,E2 -6519.251} C_VEL
LIN {X 0,Y 488.713,Z 127.607,A -85,B 0,C 180,E1 -6521.601,E2 -6521.601} C_VEL
LIN {X 0,Y 488.713,Z 127.604,A -85,B 0,C 180,E1 -6524.802,E2 -6524.802} C_VEL
LIN {X 0,Y 488.692,Z 127.609,A -85,B 0,C 180,E1 -6527.475,E2 -6527.475} C_VEL
LIN {X 0,Y 488.735,Z 127.607,A -85,B 0,C 180,E1 -6529.677,E2 -6529.677} C_VEL
LIN {X 0,Y 488.68,Z 127.611,A -85,B 0,C 180,E1 -6532.278,E2 -6532.278} C_VEL
LIN {X 0,Y 488.724,Z 127.604,A -85,B 0,C 180,E1 -6535.053,E2 -6535.053} C_VEL
LIN {X 0,Y 488.705,Z 127.609,A -85,B 0,C 180,E1 -6538.046,E2 -6538.046} C_VEL
LIN {X 0,Y 488.725,Z 127.606,A -85,B 0,C 180,E1 -6540.73,E2 -6540.73} C_VEL
LIN {X 0,Y 488.817,Z 127.708,A -85,B 0,C 180,E1 -6543.704,E2 -6543.704} C_VEL
LIN {X 0,Y 490.811,Z 137.926,A -85,B 0,C 180,E1 -6545.465,E2 -6545.465} C_VEL
LIN {X 0,Y 490.467,Z 150.431,A -85,B 0,C 180,E1 -6547.462,E2 -6547.462} C_VEL
LIN {X 0,Y 489.869,Z 167.056,A -85,B 0,C 180,E1 -6550.079,E2 -6550.079} C_VEL
LIN {X 0,Y 489.498,Z 180.89,A -85,B 0,C 180,E1 -6552.236,E2 -6552.236} C_VEL
LIN {X 0,Y 489.227,Z 190.667,A -85,B 0,C 180,E1 -6553.734,E2 -6553.734} C_VEL
LIN {X 0,Y 491.588,Z 208.169,A -85,B 0,C 180,E1 -6554.077,E2 -6554.077} C_VEL
LIN {X 0,Y 491,Z 299.872,A -85,B 0,C 180,E1 -6555.467,E2 -6555.467} C_VEL
LIN {X 0,Y 490.628,Z 312.923,A -85,B 0,C 180,E1 -6555.827,E2 -6555.827} C_VEL
LIN {X 0,Y 490.292,Z 325.003,A -85,B 0,C 180,E1 -6556.319,E2 -6556.319} C_VEL
LIN {X 0,Y 489.889,Z 336.748,A -85,B 0,C 180,E1 -6556.962,E2 -6556.962} C_VEL
LIN {X 0,Y 489.461,Z 348.178,A -85,B 0,C 180,E1 -6557.773,E2 -6557.773} C_VEL
LIN {X 0,Y 489.081,Z 358.748,A -85,B 0,C 180,E1 -6558.709,E2 -6558.709} C_VEL
LIN {X 0,Y 488.708,Z 367.388,A -85,B 0,C 180,E1 -6559.644,E2 -6559.644} C_VEL
LIN {X 0,Y 488.45,Z 375.359,A -85,B 0,C 180,E1 -6560.685,E2 -6560.685} C_VEL
LIN {X 0,Y 488.233,Z 383.153,A -85,B 0,C 180,E1 -6561.932,E2 -6561.932} C_VEL
LIN {X 0,Y 488.043,Z 390.318,A -85,B 0,C 180,E1 -6563.385,E2 -6563.385} C_VEL
LIN {X 0,Y 488.009,Z 395.092,A -85,B 0,C 180,E1 -6564.629,E2 -6564.629} C_VEL
LIN {X 0,Y 487.95,Z 398.736,A -85,B 0,C 180,E1 -6565.87,E2 -6565.87} C_VEL
LIN {X 0,Y 487.997,Z 400.619,A -85,B 0,C 180,E1 -6566.698,E2 -6566.698} C_VEL
LIN {X 0,Y 487.968,Z 402.026,A -85,B 0,C 180,E1 -6567.524,E2 -6567.524} C_VEL
LIN {X 0,Y 487.85,Z 403.628,A -85,B 0,C 180,E1 -6569.175,E2 -6569.175} C_VEL
LIN {X 0,Y 487.846,Z 403.84,A -85,B 0,C 180,E1 -6570,E2 -6570} C_VEL
LIN {X 0,Y 487.896,Z 402.992,A -85,B 0,C 180,E1 -6571.651,E2 -6571.651} C_VEL
LIN {X 0,Y 487.968,Z 401.979,A -85,B 0,C 180,E1 -6572.476,E2 -6572.476} C_VEL
LIN {X 0,Y 487.997,Z 400.557,A -85,B 0,C 180,E1 -6573.302,E2 -6573.302} C_VEL
LIN {X 0,Y 487.921,Z 397.566,A -85,B 0,C 180,E1 -6574.544,E2 -6574.544} C_VEL
LIN {X 0,Y 488.002,Z 393.531,A -85,B 0,C 180,E1 -6575.786,E2 -6575.786} C_VEL
LIN {X 0,Y 488.17,Z 387.328,A -85,B 0,C 180,E1 -6577.237,E2 -6577.237} C_VEL
LIN {X 0,Y 488.292,Z 380.554,A -85,B 0,C 180,E1 -6578.484,E2 -6578.484} C_VEL
LIN {X 0,Y 488.525,Z 372.161,A -85,B 0,C 180,E1 -6579.732,E2 -6579.732} C_VEL
LIN {X 0,Y 488.876,Z 363.55,A -85,B 0,C 180,E1 -6580.771,E2 -6580.771} C_VEL
LIN {X 0,Y 489.258,Z 352.991,A -85,B 0,C 180,E1 -6581.805,E2 -6581.805} C_VEL
LIN {X 0,Y 489.671,Z 341.62,A -85,B 0,C 180,E1 -6582.701,E2 -6582.701} C_VEL
LIN {X 0,Y 490.042,Z 330.862,A -85,B 0,C 180,E1 -6583.371,E2 -6583.371} C_VEL
LIN {X 0,Y 490.506,Z 317.618,A -85,B 0,C 180,E1 -6583.992,E2 -6583.992} C_VEL
LIN {X 0,Y 490.897,Z 304.238,A -85,B 0,C 180,E1 -6584.43,E2 -6584.43} C_VEL
LIN {X 0,Y 491.123,Z 289.179,A -85,B 0,C 180,E1 -6584.714,E2 -6584.714} C_VEL
LIN {X 0,Y 491.473,Z 206.775,A -85,B 0,C 180,E1 -6585.953,E2 -6585.953} C_VEL
LIN {X 0,Y 489.194,Z 189.826,A -85,B 0,C 180,E1 -6586.3,E2 -6586.3} C_VEL
LIN {X 0,Y 489.73,Z 169.094,A -85,B 0,C 180,E1 -6589.491,E2 -6589.491} C_VEL
LIN {X 0,Y 490.204,Z 152.269,A -85,B 0,C 180,E1 -6592.107,E2 -6592.107} C_VEL
LIN {X 0,Y 490.655,Z 138.232,A -85,B 0,C 180,E1 -6594.318,E2 -6594.318} C_VEL
LIN {X 0,Y 489.236,Z 129.69,A -85,B 0,C 180,E1 -6595.756,E2 -6595.756} C_VEL
LIN {X 0,Y 488.786,Z 127.603,A -85,B 0,C 180,E1 -6596.125,E2 -6596.125} C_VEL
LIN {X 0,Y 488.725,Z 127.607,A -85,B 0,C 180,E1 -6599.27,E2 -6599.27} C_VEL
LIN {X 0,Y 488.704,Z 127.613,A -85,B 0,C 180,E1 -6602.147,E2 -6602.147} C_VEL
LIN {X 0,Y 488.718,Z 127.606,A -85,B 0,C 180,E1 -6605.115,E2 -6605.115} C_VEL
LIN {X 0,Y 488.684,Z 127.619,A -85,B 0,C 180,E1 -6608.199,E2 -6608.199} C_VEL
LIN {X 0,Y 488.75,Z 127.608,A -85,B 0,C 180,E1 -6610.349,E2 -6610.349} C_VEL
LIN {X 0,Y 488.687,Z 127.612,A -85,B 0,C 180,E1 -6613.654,E2 -6613.654} C_VEL
LIN {X 0,Y 488.687,Z 127.614,A -85,B 0,C 180,E1 -6616.345,E2 -6616.345} C_VEL
LIN {X 0,Y 488.733,Z 127.607,A -85,B 0,C 180,E1 -6619.676,E2 -6619.676} C_VEL
LIN {X 0,Y 488.678,Z 127.613,A -85,B 0,C 180,E1 -6622.278,E2 -6622.278} C_VEL
LIN {X 0,Y 488.722,Z 127.604,A -85,B 0,C 180,E1 -6625.052,E2 -6625.052} C_VEL
LIN {X 0,Y 488.702,Z 127.611,A -85,B 0,C 180,E1 -6628.046,E2 -6628.046} C_VEL
LIN {X 0,Y 488.722,Z 127.601,A -85,B 0,C 180,E1 -6630.729,E2 -6630.729} C_VEL
LIN {X 0,Y 488.752,Z 127.605,A -85,B 0,C 180,E1 -6633.528,E2 -6633.528} C_VEL
LIN {X 0,Y 488.678,Z 127.608,A -85,B 0,C 180,E1 -6636.254,E2 -6636.254} C_VEL
LIN {X 0,Y 488.745,Z 127.603,A -85,B 0,C 180,E1 -6639.175,E2 -6639.175} C_VEL
LIN {X 0,Y 488.758,Z 127.604,A -85,B 0,C 180,E1 -6641.627,E2 -6641.627} C_VEL
LIN {X 0,Y 488.763,Z 127.599,A -85,B 0,C 180,E1 -6644.999,E2 -6644.999} C_VEL
LIN {X 0,Y 488.804,Z 127.591,A -85,B 0,C 180,E1 -6648.387,E2 -6648.387} C_VEL
LIN {X 0,Y 488.816,Z 127.592,A -85,B 0,C 180,E1 -6651.733,E2 -6651.733} C_VEL
LIN {X 0,Y 488.856,Z 127.587,A -85,B 0,C 180,E1 -6654.224,E2 -6654.224} C_VEL
LIN {X 0,Y 488.96,Z 127.577,A -85,B 0,C 180,E1 -6657.528,E2 -6657.528} C_VEL
LIN {X 0,Y 488.952,Z 127.579,A -85,B 0,C 180,E1 -6660.823,E2 -6660.823} C_VEL
LIN {X 0,Y 488.96,Z 127.576,A -85,B 0,C 180,E1 -6662.471,E2 -6662.471} C_VEL
LIN {X 0,Y 488.846,Z 127.587,A -85,B 0,C 180,E1 -6665.776,E2 -6665.776} C_VEL
LIN {X 0,Y 488.815,Z 127.594,A -85,B 0,C 180,E1 -6668.266,E2 -6668.266} C_VEL
LIN {X 0,Y 488.803,Z 127.593,A -85,B 0,C 180,E1 -6671.612,E2 -6671.612} C_VEL
LIN {X 0,Y 488.759,Z 127.604,A -85,B 0,C 180,E1 -6675,E2 -6675} C_VEL
LIN {X 0,Y 488.753,Z 127.605,A -85,B 0,C 180,E1 -6678.442,E2 -6678.442} C_VEL
LIN {X 0,Y 488.704,Z 127.609,A -85,B 0,C 180,E1 -6681.071,E2 -6681.071} C_VEL
LIN {X 0,Y 488.686,Z 127.612,A -85,B 0,C 180,E1 -6683.746,E2 -6683.746} C_VEL
LIN {X 0,Y 488.79,Z 127.601,A -85,B 0,C 180,E1 -6686.944,E2 -6686.944} C_VEL
LIN {X 0,Y 488.708,Z 127.613,A -85,B 0,C 180,E1 -6690.363,E2 -6690.363} C_VEL
LIN {X 0,Y 488.734,Z 127.607,A -85,B 0,C 180,E1 -6693.485,E2 -6693.485} C_VEL
LIN {X 0,Y 488.827,Z 127.779,A -85,B 0,C 180,E1 -6694.167,E2 -6694.167} C_VEL
LIN {X 0,Y 489.567,Z 133.243,A -85,B 0,C 180,E1 -6695.296,E2 -6695.296} C_VEL
LIN {X 0,Y 489.481,Z 140.653,A -85,B 0,C 180,E1 -6696.779,E2 -6696.779} C_VEL
LIN {X 0,Y 491.814,Z 151.689,A -85,B 0,C 180,E1 -6697.043,E2 -6697.043} C_VEL
LIN {X 0,Y 491.158,Z 248.226,A -85,B 0,C 180,E1 -6698.519,E2 -6698.519} C_VEL
LIN {X 0,Y 490.911,Z 261.885,A -85,B 0,C 180,E1 -6698.909,E2 -6698.909} C_VEL
LIN {X 0,Y 490.65,Z 274.571,A -85,B 0,C 180,E1 -6699.453,E2 -6699.453} C_VEL
LIN {X 0,Y 490.303,Z 286.821,A -85,B 0,C 180,E1 -6700.168,E2 -6700.168} C_VEL
LIN {X 0,Y 489.954,Z 297.756,A -85,B 0,C 180,E1 -6700.984,E2 -6700.984} C_VEL
LIN {X 0,Y 489.534,Z 307.864,A -85,B 0,C 180,E1 -6701.924,E2 -6701.924} C_VEL
LIN {X 0,Y 489.144,Z 317.919,A -85,B 0,C 180,E1 -6703.094,E2 -6703.094} C_VEL
LIN {X 0,Y 488.759,Z 325.972,A -85,B 0,C 180,E1 -6704.249,E2 -6704.249} C_VEL
LIN {X 0,Y 488.565,Z 330.874,A -85,B 0,C 180,E1 -6705.095,E2 -6705.095} C_VEL
LIN {X 0,Y 487.787,Z 333.974,A -85,B 0,C 180,E1 -6705.681,E2 -6705.681} C_VEL
LIN {X 0,Y 484.77,Z 338.6,A -85,B 0,C 180,E1 -6706.652,E2 -6706.652} C_VEL
LIN {X 0,Y 481.769,Z 342.545,A -85,B 0,C 180,E1 -6707.672,E2 -6707.672} C_VEL
LIN {X 0,Y 481.029,Z 344.512,A -85,B 0,C 180,E1 -6708.331,E2 -6708.331} C_VEL
LIN {X 0,Y 480.93,Z 347.235,A -85,B 0,C 180,E1 -6709.455,E2 -6709.455} C_VEL
LIN {X 0,Y 480.824,Z 349.781,A -85,B 0,C 180,E1 -6711.06,E2 -6711.06} C_VEL
LIN {X 0,Y 480.787,Z 350.613,A -85,B 0,C 180,E1 -6712.125,E2 -6712.125} C_VEL
LIN {X 0,Y 480.773,Z 350.769,A -85,B 0,C 180,E1 -6713.513,E2 -6713.513} C_VEL
LIN {X 0,Y 480.821,Z 349.805,A -85,B 0,C 180,E1 -6714.938,E2 -6714.938} C_VEL
LIN {X 0,Y 480.938,Z 347.606,A -85,B 0,C 180,E1 -6716.403,E2 -6716.403} C_VEL
LIN {X 0,Y 481.071,Z 343.924,A -85,B 0,C 180,E1 -6717.922,E2 -6717.922} C_VEL
LIN {X 0,Y 481.199,Z 339.447,A -85,B 0,C 180,E1 -6719.258,E2 -6719.258} C_VEL
LIN {X 0,Y 481.451,Z 333.034,A -85,B 0,C 180,E1 -6720.723,E2 -6720.723} C_VEL
LIN {X 0,Y 481.757,Z 326.277,A -85,B 0,C 180,E1 -6721.935,E2 -6721.935} C_VEL
LIN {X 0,Y 482.098,Z 318.022,A -85,B 0,C 180,E1 -6723.134,E2 -6723.134} C_VEL
LIN {X 0,Y 482.495,Z 308.835,A -85,B 0,C 180,E1 -6724.22,E2 -6724.22} C_VEL
LIN {X 0,Y 482.948,Z 297.822,A -85,B 0,C 180,E1 -6725.268,E2 -6725.268} C_VEL
LIN {X 0,Y 483.377,Z 286.957,A -85,B 0,C 180,E1 -6726.086,E2 -6726.086} C_VEL
LIN {X 0,Y 483.72,Z 274.55,A -85,B 0,C 180,E1 -6726.82,E2 -6726.82} C_VEL
LIN {X 0,Y 484.01,Z 263.39,A -85,B 0,C 180,E1 -6727.313,E2 -6727.313} C_VEL
LIN {X 0,Y 484.234,Z 250.159,A -85,B 0,C 180,E1 -6727.718,E2 -6727.718} C_VEL
LIN {X 0,Y 484.423,Z 230.448,A -85,B 0,C 180,E1 -6728.057,E2 -6728.057} C_VEL
LIN {X 0,Y 484.872,Z 152.697,A -85,B 0,C 180,E1 -6729.241,E2 -6729.241} C_VEL
LIN {X 0,Y 482.362,Z 140.504,A -85,B 0,C 180,E1 -6729.533,E2 -6729.533} C_VEL
LIN {X 0,Y 482.464,Z 133.839,A -85,B 0,C 180,E1 -6730.912,E2 -6730.912} C_VEL
LIN {X 0,Y 481.729,Z 128.482,A -85,B 0,C 180,E1 -6732.07,E2 -6732.07} C_VEL
LIN {X 0,Y 481.742,Z 128.475,A -85,B 0,C 180,E1 -6734.776,E2 -6734.776} C_VEL
LIN {X 0,Y 481.751,Z 128.473,A -85,B 0,C 180,E1 -6738.215,E2 -6738.215} C_VEL
LIN {X 0,Y 481.761,Z 128.478,A -85,B 0,C 180,E1 -6741.612,E2 -6741.612} C_VEL
LIN {X 0,Y 481.808,Z 128.465,A -85,B 0,C 180,E1 -6744.14,E2 -6744.14} C_VEL
LIN {X 0,Y 481.928,Z 128.457,A -85,B 0,C 180,E1 -6747.493,E2 -6747.493} C_VEL
LIN {X 0,Y 481.886,Z 128.457,A -85,B 0,C 180,E1 -6750.836,E2 -6750.836} C_VEL
LIN {X 0,Y 481.928,Z 128.45,A -85,B 0,C 180,E1 -6752.507,E2 -6752.507} C_VEL
LIN {X 0,Y 481.801,Z 128.466,A -85,B 0,C 180,E1 -6755.861,E2 -6755.861} C_VEL
LIN {X 0,Y 481.74,Z 128.473,A -85,B 0,C 180,E1 -6758.389,E2 -6758.389} C_VEL
LIN {X 0,Y 481.751,Z 128.472,A -85,B 0,C 180,E1 -6761.785,E2 -6761.785} C_VEL
LIN {X 0,Y 481.743,Z 128.477,A -85,B 0,C 180,E1 -6765.224,E2 -6765.224} C_VEL
LIN {X 0,Y 481.708,Z 128.483,A -85,B 0,C 180,E1 -6768.722,E2 -6768.722} C_VEL
LIN {X 0,Y 481.645,Z 128.486,A -85,B 0,C 180,E1 -6771.395,E2 -6771.395} C_VEL
LIN {X 0,Y 481.673,Z 128.482,A -85,B 0,C 180,E1 -6774.113,E2 -6774.113} C_VEL
LIN {X 0,Y 481.746,Z 128.474,A -85,B 0,C 180,E1 -6777.139,E2 -6777.139} C_VEL
LIN {X 0,Y 481.678,Z 128.481,A -85,B 0,C 180,E1 -6779.741,E2 -6779.741} C_VEL
LIN {X 0,Y 481.669,Z 128.488,A -85,B 0,C 180,E1 -6782.674,E2 -6782.674} C_VEL
LIN {X 0,Y 481.635,Z 128.486,A -85,B 0,C 180,E1 -6785.709,E2 -6785.709} C_VEL
LIN {X 0,Y 481.669,Z 128.484,A -85,B 0,C 180,E1 -6788.859,E2 -6788.859} C_VEL
LIN {X 0,Y 481.651,Z 128.487,A -85,B 0,C 180,E1 -6791.913,E2 -6791.913} C_VEL
LIN {X 0,Y 481.658,Z 128.488,A -85,B 0,C 180,E1 -6794.457,E2 -6794.457} C_VEL
LIN {X 0,Y 481.646,Z 128.488,A -85,B 0,C 180,E1 -6797.839,E2 -6797.839} C_VEL
LIN {X 0,Y 481.679,Z 128.482,A -85,B 0,C 180,E1 -6800.651,E2 -6800.651} C_VEL
LIN {X 0,Y 481.628,Z 128.488,A -85,B 0,C 180,E1 -6803.376,E2 -6803.376} C_VEL
LIN {X 0,Y 481.708,Z 128.48,A -85,B 0,C 180,E1 -6806.33,E2 -6806.33} C_VEL
LIN {X 0,Y 481.65,Z 128.486,A -85,B 0,C 180,E1 -6809.417,E2 -6809.417} C_VEL
LIN {X 0,Y 481.698,Z 128.481,A -85,B 0,C 180,E1 -6812.168,E2 -6812.168} C_VEL
LIN {X 0,Y 481.691,Z 128.479,A -85,B 0,C 180,E1 -6814.969,E2 -6814.969} C_VEL
LIN {X 0,Y 481.647,Z 128.492,A -85,B 0,C 180,E1 -6817.705,E2 -6817.705} C_VEL
LIN {X 0,Y 481.704,Z 128.478,A -85,B 0,C 180,E1 -6820.393,E2 -6820.393} C_VEL
LIN {X 0,Y 481.689,Z 128.481,A -85,B 0,C 180,E1 -6823.034,E2 -6823.034} C_VEL
LIN {X 0,Y 481.692,Z 128.484,A -85,B 0,C 180,E1 -6825.639,E2 -6825.639} C_VEL
LIN {X 0,Y 481.749,Z 128.472,A -85,B 0,C 180,E1 -6828.215,E2 -6828.215} C_VEL
LIN {X 0,Y 481.762,Z 128.474,A -85,B 0,C 180,E1 -6831.612,E2 -6831.612} C_VEL
LIN {X 0,Y 481.817,Z 128.463,A -85,B 0,C 180,E1 -6834.14,E2 -6834.14} C_VEL
LIN {X 0,Y 481.927,Z 128.453,A -85,B 0,C 180,E1 -6837.493,E2 -6837.493} C_VEL
LIN {X 0,Y 481.904,Z 128.457,A -85,B 0,C 180,E1 -6840.836,E2 -6840.836} C_VEL
LIN {X 0,Y 481.927,Z 128.451,A -85,B 0,C 180,E1 -6842.508,E2 -6842.508} C_VEL
LIN {X 0,Y 481.807,Z 128.464,A -85,B 0,C 180,E1 -6845.861,E2 -6845.861} C_VEL
LIN {X 0,Y 481.761,Z 128.472,A -85,B 0,C 180,E1 -6848.389,E2 -6848.389} C_VEL
LIN {X 0,Y 481.75,Z 128.471,A -85,B 0,C 180,E1 -6851.785,E2 -6851.785} C_VEL
LIN {X 0,Y 481.741,Z 128.475,A -85,B 0,C 180,E1 -6855.224,E2 -6855.224} C_VEL
LIN {X 0,Y 481.712,Z 128.483,A -85,B 0,C 180,E1 -6858.722,E2 -6858.722} C_VEL
LIN {X 0,Y 481.644,Z 128.485,A -85,B 0,C 180,E1 -6861.395,E2 -6861.395} C_VEL
LIN {X 0,Y 481.673,Z 128.484,A -85,B 0,C 180,E1 -6864.114,E2 -6864.114} C_VEL
LIN {X 0,Y 481.746,Z 128.473,A -85,B 0,C 180,E1 -6867.139,E2 -6867.139} C_VEL
LIN {X 0,Y 481.678,Z 128.482,A -85,B 0,C 180,E1 -6869.741,E2 -6869.741} C_VEL
LIN {X 0,Y 481.671,Z 128.484,A -85,B 0,C 180,E1 -6872.674,E2 -6872.674} C_VEL
LIN {X 0,Y 481.636,Z 128.488,A -85,B 0,C 180,E1 -6875.71,E2 -6875.71} C_VEL
LIN {X 0,Y 481.715,Z 128.476,A -85,B 0,C 180,E1 -6879.354,E2 -6879.354} C_VEL
LIN {X 0,Y 481.649,Z 128.491,A -85,B 0,C 180,E1 -6882.161,E2 -6882.161} C_VEL
LIN {X 0,Y 481.66,Z 128.485,A -85,B 0,C 180,E1 -6885.543,E2 -6885.543} C_VEL
LIN {X 0,Y 481.669,Z 128.482,A -85,B 0,C 180,E1 -6888.96,E2 -6888.96} C_VEL
LIN {X 0,Y 481.699,Z 128.479,A -85,B 0,C 180,E1 -6891.144,E2 -6891.144} C_VEL
LIN {X 0,Y 481.663,Z 128.482,A -85,B 0,C 180,E1 -6894.796,E2 -6894.796} C_VEL
LIN {X 0,Y 481.673,Z 128.485,A -85,B 0,C 180,E1 -6897.326,E2 -6897.326} C_VEL
LIN {X 0,Y 481.681,Z 128.485,A -85,B 0,C 180,E1 -6900.259,E2 -6900.259} C_VEL
LIN {X 0,Y 481.766,Z 128.519,A -85,B 0,C 180,E1 -6903.494,E2 -6903.494} C_VEL
LIN {X 0,Y 483.809,Z 138.922,A -85,B 0,C 180,E1 -6905.315,E2 -6905.315} C_VEL
LIN {X 0,Y 483.699,Z 147.62,A -85,B 0,C 180,E1 -6906.734,E2 -6906.734} C_VEL
LIN {X 0,Y 482.971,Z 165.279,A -85,B 0,C 180,E1 -6909.559,E2 -6909.559} C_VEL
LIN {X 0,Y 482.601,Z 179.117,A -85,B 0,C 180,E1 -6911.754,E2 -6911.754} C_VEL
LIN {X 0,Y 482.234,Z 190.268,A -85,B 0,C 180,E1 -6913.496,E2 -6913.496} C_VEL
LIN {X 0,Y 484.757,Z 209.424,A -85,B 0,C 180,E1 -6913.877,E2 -6913.877} C_VEL
LIN {X 0,Y 484.131,Z 299.208,A -85,B 0,C 180,E1 -6915.256,E2 -6915.256} C_VEL
LIN {X 0,Y 483.762,Z 312.351,A -85,B 0,C 180,E1 -6915.621,E2 -6915.621} C_VEL
LIN {X 0,Y 483.337,Z 325.595,A -85,B 0,C 180,E1 -6916.172,E2 -6916.172} C_VEL
LIN {X 0,Y 482.884,Z 338.016,A -85,B 0,C 180,E1 -6916.888,E2 -6916.888} C_VEL
LIN {X 0,Y 482.441,Z 348.918,A -85,B 0,C 180,E1 -6917.691,E2 -6917.691} C_VEL
LIN {X 0,Y 482.04,Z 359.373,A -85,B 0,C 180,E1 -6918.649,E2 -6918.649} C_VEL
LIN {X 0,Y 481.632,Z 368.672,A -85,B 0,C 180,E1 -6919.703,E2 -6919.703} C_VEL
LIN {X 0,Y 481.307,Z 377.714,A -85,B 0,C 180,E1 -6920.969,E2 -6920.969} C_VEL
LIN {X 0,Y 481.087,Z 385,A -85,B 0,C 180,E1 -6922.234,E2 -6922.234} C_VEL
LIN {X 0,Y 480.933,Z 391.095,A -85,B 0,C 180,E1 -6923.568,E2 -6923.568} C_VEL
LIN {X 0,Y 480.894,Z 396.026,A -85,B 0,C 180,E1 -6924.969,E2 -6924.969} C_VEL
LIN {X 0,Y 480.847,Z 398.343,A -85,B 0,C 180,E1 -6925.809,E2 -6925.809} C_VEL
LIN {X 0,Y 480.919,Z 400.229,A -85,B 0,C 180,E1 -6926.649,E2 -6926.649} C_VEL
LIN {X 0,Y 480.879,Z 401.638,A -85,B 0,C 180,E1 -6927.487,E2 -6927.487} C_VEL
LIN {X 0,Y 480.827,Z 402.636,A -85,B 0,C 180,E1 -6928.325,E2 -6928.325} C_VEL
LIN {X 0,Y 480.768,Z 403.452,A -85,B 0,C 180,E1 -6930,E2 -6930} C_VEL
LIN {X 0,Y 480.828,Z 402.603,A -85,B 0,C 180,E1 -6931.675,E2 -6931.675} C_VEL
LIN {X 0,Y 480.879,Z 401.588,A -85,B 0,C 180,E1 -6932.513,E2 -6932.513} C_VEL
LIN {X 0,Y 480.919,Z 400.165,A -85,B 0,C 180,E1 -6933.351,E2 -6933.351} C_VEL
LIN {X 0,Y 480.839,Z 397.172,A -85,B 0,C 180,E1 -6934.611,E2 -6934.611} C_VEL
LIN {X 0,Y 480.899,Z 393.133,A -85,B 0,C 180,E1 -6935.872,E2 -6935.872} C_VEL
LIN {X 0,Y 481.095,Z 386.928,A -85,B 0,C 180,E1 -6937.344,E2 -6937.344} C_VEL
LIN {X 0,Y 481.234,Z 380.151,A -85,B 0,C 180,E1 -6938.609,E2 -6938.609} C_VEL
LIN {X 0,Y 481.484,Z 371.752,A -85,B 0,C 180,E1 -6939.875,E2 -6939.875} C_VEL
LIN {X 0,Y 481.858,Z 363.137,A -85,B 0,C 180,E1 -6940.93,E2 -6940.93} C_VEL
LIN {X 0,Y 482.255,Z 352.797,A -85,B 0,C 180,E1 -6941.959,E2 -6941.959} C_VEL
LIN {X 0,Y 482.672,Z 342.285,A -85,B 0,C 180,E1 -6942.808,E2 -6942.808} C_VEL
LIN {X 0,Y 483.128,Z 330.453,A -85,B 0,C 180,E1 -6943.566,E2 -6943.566} C_VEL
LIN {X 0,Y 483.567,Z 318.521,A -85,B 0,C 180,E1 -6944.143,E2 -6944.143} C_VEL
LIN {X 0,Y 483.98,Z 305.688,A -85,B 0,C 180,E1 -6944.587,E2 -6944.587} C_VEL
LIN {X 0,Y 484.246,Z 292.38,A -85,B 0,C 180,E1 -6944.874,E2 -6944.874} C_VEL
LIN {X 0,Y 484.628,Z 207.382,A -85,B 0,C 180,E1 -6946.172,E2 -6946.172} C_VEL
LIN {X 0,Y 482.199,Z 189.46,A -85,B 0,C 180,E1 -6946.539,E2 -6946.539} C_VEL
LIN {X 0,Y 482.776,Z 168.697,A -85,B 0,C 180,E1 -6949.783,E2 -6949.783} C_VEL
LIN {X 0,Y 483.392,Z 150.498,A -85,B 0,C 180,E1 -6952.661,E2 -6952.661} C_VEL
LIN {X 0,Y 483.7,Z 139.261,A -85,B 0,C 180,E1 -6954.462,E2 -6954.462} C_VEL
LIN {X 0,Y 482.21,Z 130.713,A -85,B 0,C 180,E1 -6955.927,E2 -6955.927} C_VEL
LIN {X 0,Y 481.752,Z 128.48,A -85,B 0,C 180,E1 -6956.361,E2 -6956.361} C_VEL
LIN {X 0,Y 481.68,Z 128.486,A -85,B 0,C 180,E1 -6959.741,E2 -6959.741} C_VEL
LIN {X 0,Y 481.673,Z 128.488,A -85,B 0,C 180,E1 -6962.674,E2 -6962.674} C_VEL
LIN {X 0,Y 481.638,Z 128.49,A -85,B 0,C 180,E1 -6965.709,E2 -6965.709} C_VEL
LIN {X 0,Y 481.715,Z 128.479,A -85,B 0,C 180,E1 -6969.353,E2 -6969.353} C_VEL
LIN {X 0,Y 481.649,Z 128.495,A -85,B 0,C 180,E1 -6972.16,E2 -6972.16} C_VEL
LIN {X 0,Y 481.66,Z 128.488,A -85,B 0,C 180,E1 -6975.542,E2 -6975.542} C_VEL
LIN {X 0,Y 481.668,Z 128.483,A -85,B 0,C 180,E1 -6978.959,E2 -6978.959} C_VEL
LIN {X 0,Y 481.697,Z 128.478,A -85,B 0,C 180,E1 -6981.143,E2 -6981.143} C_VEL
LIN {X 0,Y 481.661,Z 128.483,A -85,B 0,C 180,E1 -6984.795,E2 -6984.795} C_VEL
LIN {X 0,Y 481.671,Z 128.483,A -85,B 0,C 180,E1 -6987.325,E2 -6987.325} C_VEL
LIN {X 0,Y 481.678,Z 128.481,A -85,B 0,C 180,E1 -6990.259,E2 -6990.259} C_VEL
LIN {X 0,Y 481.744,Z 128.474,A -85,B 0,C 180,E1 -6993.112,E2 -6993.112} C_VEL
LIN {X 0,Y 481.659,Z 128.486,A -85,B 0,C 180,E1 -6995.886,E2 -6995.886} C_VEL
LIN {X 0,Y 481.701,Z 128.479,A -85,B 0,C 180,E1 -6999.027,E2 -6999.027} C_VEL
LIN {X 0,Y 481.706,Z 128.477,A -85,B 0,C 180,E1 -7002.158,E2 -7002.158} C_VEL
LIN {X 0,Y 481.743,Z 128.472,A -85,B 0,C 180,E1 -7004.776,E2 -7004.776} C_VEL
LIN {X 0,Y 481.749,Z 128.47,A -85,B 0,C 180,E1 -7008.215,E2 -7008.215} C_VEL
LIN {X 0,Y 481.761,Z 128.472,A -85,B 0,C 180,E1 -7011.611,E2 -7011.611} C_VEL
LIN {X 0,Y 481.817,Z 128.464,A -85,B 0,C 180,E1 -7014.139,E2 -7014.139} C_VEL
LIN {X 0,Y 481.927,Z 128.454,A -85,B 0,C 180,E1 -7017.492,E2 -7017.492} C_VEL
LIN {X 0,Y 481.903,Z 128.457,A -85,B 0,C 180,E1 -7020.835,E2 -7020.835} C_VEL
LIN {X 0,Y 481.927,Z 128.452,A -85,B 0,C 180,E1 -7022.507,E2 -7022.507} C_VEL
LIN {X 0,Y 481.806,Z 128.464,A -85,B 0,C 180,E1 -7025.86,E2 -7025.86} C_VEL
LIN {X 0,Y 481.76,Z 128.474,A -85,B 0,C 180,E1 -7028.388,E2 -7028.388} C_VEL
LIN {X 0,Y 481.749,Z 128.472,A -85,B 0,C 180,E1 -7031.785,E2 -7031.785} C_VEL
LIN {X 0,Y 481.74,Z 128.476,A -85,B 0,C 180,E1 -7035.224,E2 -7035.224} C_VEL
LIN {X 0,Y 481.71,Z 128.485,A -85,B 0,C 180,E1 -7038.722,E2 -7038.722} C_VEL
LIN {X 0,Y 481.643,Z 128.487,A -85,B 0,C 180,E1 -7041.395,E2 -7041.395} C_VEL
LIN {X 0,Y 481.671,Z 128.489,A -85,B 0,C 180,E1 -7044.113,E2 -7044.113} C_VEL
LIN {X 0,Y 481.745,Z 128.477,A -85,B 0,C 180,E1 -7047.139,E2 -7047.139} C_VEL
LIN {X 0,Y 481.677,Z 128.484,A -85,B 0,C 180,E1 -7049.741,E2 -7049.741} C_VEL
LIN {X 0,Y 481.673,Z 128.489,A -85,B 0,C 180,E1 -7052.674,E2 -7052.674} C_VEL
LIN {X 0,Y 481.742,Z 128.513,A -85,B 0,C 180,E1 -7053.963,E2 -7053.963} C_VEL
LIN {X 0,Y 482.596,Z 133.387,A -85,B 0,C 180,E1 -7054.988,E2 -7054.988} C_VEL
LIN {X 0,Y 482.547,Z 141.056,A -85,B 0,C 180,E1 -7056.535,E2 -7056.535} C_VEL
LIN {X 0,Y 485.051,Z 153.08,A -85,B 0,C 180,E1 -7056.824,E2 -7056.824} C_VEL
LIN {X 0,Y 484.315,Z 248.58,A -85,B 0,C 180,E1 -7058.306,E2 -7058.306} C_VEL
LIN {X 0,Y 484.063,Z 262.106,A -85,B 0,C 180,E1 -7058.698,E2 -7058.698} C_VEL
LIN {X 0,Y 483.818,Z 273.655,A -85,B 0,C 180,E1 -7059.189,E2 -7059.189} C_VEL
LIN {X 0,Y 483.47,Z 285.994,A -85,B 0,C 180,E1 -7059.898,E2 -7059.898} C_VEL
LIN {X 0,Y 483.055,Z 297.525,A -85,B 0,C 180,E1 -7060.756,E2 -7060.756} C_VEL
LIN {X 0,Y 482.583,Z 308.22,A -85,B 0,C 180,E1 -7061.756,E2 -7061.756} C_VEL
LIN {X 0,Y 482.172,Z 318.031,A -85,B 0,C 180,E1 -7062.91,E2 -7062.91} C_VEL
LIN {X 0,Y 481.767,Z 326.076,A -85,B 0,C 180,E1 -7064.073,E2 -7064.073} C_VEL
LIN {X 0,Y 481.483,Z 332.717,A -85,B 0,C 180,E1 -7065.253,E2 -7065.253} C_VEL
LIN {X 0,Y 481.236,Z 338.977,A -85,B 0,C 180,E1 -7066.655,E2 -7066.655} C_VEL
LIN {X 0,Y 481.05,Z 344.08,A -85,B 0,C 180,E1 -7068.167,E2 -7068.167} C_VEL
LIN {X 0,Y 481.029,Z 344.512,A -85,B 0,C 180,E1 -7068.331,E2 -7068.331} C_VEL
LIN {X 0,Y 480.298,Z 346.312,A -85,B 0,C 180,E1 -7068.999,E2 -7068.999} C_VEL
LIN {X 0,Y 477.341,Z 348.672,A -85,B 0,C 180,E1 -7070.095,E2 -7070.095} C_VEL
LIN {X 0,Y 474.863,Z 350.095,A -85,B 0,C 180,E1 -7070.991,E2 -7070.991} C_VEL
LIN {X 0,Y 473.786,Z 350.768,A -85,B 0,C 180,E1 -7071.691,E2 -7071.691} C_VEL
LIN {X 0,Y 473.691,Z 350.898,A -85,B 0,C 180,E1 -7071.929,E2 -7071.929} C_VEL
LIN {X 0,Y 473.697,Z 351.139,A -85,B 0,C 180,E1 -7073.597,E2 -7073.597} C_VEL
LIN {X 0,Y 473.71,Z 350.456,A -85,B 0,C 180,E1 -7074.685,E2 -7074.685} C_VEL
LIN {X 0,Y 473.819,Z 348.488,A -85,B 0,C 180,E1 -7076.163,E2 -7076.163} C_VEL
LIN {X 0,Y 473.965,Z 345.028,A -85,B 0,C 180,E1 -7077.737,E2 -7077.737} C_VEL
LIN {X 0,Y 474.131,Z 340.047,A -85,B 0,C 180,E1 -7079.286,E2 -7079.286} C_VEL
LIN {X 0,Y 474.393,Z 333.871,A -85,B 0,C 180,E1 -7080.733,E2 -7080.733} C_VEL
LIN {X 0,Y 474.722,Z 327.236,A -85,B 0,C 180,E1 -7081.964,E2 -7081.964} C_VEL
LIN {X 0,Y 475.088,Z 319.115,A -85,B 0,C 180,E1 -7083.18,E2 -7083.18} C_VEL
LIN {X 0,Y 475.53,Z 309.356,A -85,B 0,C 180,E1 -7084.36,E2 -7084.36} C_VEL
LIN {X 0,Y 475.978,Z 299.27,A -85,B 0,C 180,E1 -7085.347,E2 -7085.347} C_VEL
LIN {X 0,Y 476.372,Z 288.927,A -85,B 0,C 180,E1 -7086.162,E2 -7086.162} C_VEL
LIN {X 0,Y 476.731,Z 277.227,A -85,B 0,C 180,E1 -7086.89,E2 -7086.89} C_VEL
LIN {X 0,Y 477.113,Z 264.558,A -85,B 0,C 180,E1 -7087.481,E2 -7087.481} C_VEL
LIN {X 0,Y 477.363,Z 251.727,A -85,B 0,C 180,E1 -7087.896,E2 -7087.896} C_VEL
LIN {X 0,Y 477.527,Z 235.791,A -85,B 0,C 180,E1 -7088.192,E2 -7088.192} C_VEL
LIN {X 0,Y 478.119,Z 153.969,A -85,B 0,C 180,E1 -7089.455,E2 -7089.455} C_VEL
LIN {X 0,Y 475.422,Z 140.937,A -85,B 0,C 180,E1 -7089.757,E2 -7089.757} C_VEL
LIN {X 0,Y 475.444,Z 134.54,A -85,B 0,C 180,E1 -7091.093,E2 -7091.093} C_VEL
LIN {X 0,Y 474.691,Z 129.358,A -85,B 0,C 180,E1 -7092.22,E2 -7092.22} C_VEL
LIN {X 0,Y 474.648,Z 129.363,A -85,B 0,C 180,E1 -7095.421,E2 -7095.421} C_VEL
LIN {X 0,Y 474.704,Z 129.352,A -85,B 0,C 180,E1 -7098.038,E2 -7098.038} C_VEL
LIN {X 0,Y 474.726,Z 129.354,A -85,B 0,C 180,E1 -7101.487,E2 -7101.487} C_VEL
LIN {X 0,Y 474.771,Z 129.343,A -85,B 0,C 180,E1 -7104.052,E2 -7104.052} C_VEL
LIN {X 0,Y 474.894,Z 129.333,A -85,B 0,C 180,E1 -7107.455,E2 -7107.455} C_VEL
LIN {X 0,Y 474.912,Z 129.324,A -85,B 0,C 180,E1 -7110,E2 -7110} C_VEL
LIN {X 0,Y 474.894,Z 129.326,A -85,B 0,C 180,E1 -7112.545,E2 -7112.545} C_VEL
LIN {X 0,Y 474.762,Z 129.343,A -85,B 0,C 180,E1 -7115.948,E2 -7115.948} C_VEL
LIN {X 0,Y 474.711,Z 129.349,A -85,B 0,C 180,E1 -7118.514,E2 -7118.514} C_VEL
LIN {X 0,Y 474.705,Z 129.349,A -85,B 0,C 180,E1 -7121.962,E2 -7121.962} C_VEL
LIN {X 0,Y 474.7,Z 129.352,A -85,B 0,C 180,E1 -7125.456,E2 -7125.456} C_VEL
LIN {X 0,Y 474.662,Z 129.361,A -85,B 0,C 180,E1 -7129.01,E2 -7129.01} C_VEL
LIN {X 0,Y 474.588,Z 129.364,A -85,B 0,C 180,E1 -7131.729,E2 -7131.729} C_VEL
LIN {X 0,Y 474.655,Z 129.36,A -85,B 0,C 180,E1 -7134.493,E2 -7134.493} C_VEL
LIN {X 0,Y 474.68,Z 129.353,A -85,B 0,C 180,E1 -7137.334,E2 -7137.334} C_VEL
LIN {X 0,Y 474.603,Z 129.367,A -85,B 0,C 180,E1 -7140.81,E2 -7140.81} C_VEL
LIN {X 0,Y 474.624,Z 129.36,A -85,B 0,C 180,E1 -7143.221,E2 -7143.221} C_VEL
LIN {X 0,Y 474.588,Z 129.37,A -85,B 0,C 180,E1 -7146.323,E2 -7146.323} C_VEL
LIN {X 0,Y 474.616,Z 129.361,A -85,B 0,C 180,E1 -7149.646,E2 -7149.646} C_VEL
LIN {X 0,Y 474.613,Z 129.361,A -85,B 0,C 180,E1 -7152.934,E2 -7152.934} C_VEL
LIN {X 0,Y 474.608,Z 129.365,A -85,B 0,C 180,E1 -7155.895,E2 -7155.895} C_VEL
LIN {X 0,Y 474.626,Z 129.359,A -85,B 0,C 180,E1 -7159.041,E2 -7159.041} C_VEL
LIN {X 0,Y 474.609,Z 129.365,A -85,B 0,C 180,E1 -7161.704,E2 -7161.704} C_VEL
LIN {X 0,Y 474.627,Z 129.359,A -85,B 0,C 180,E1 -7164.726,E2 -7164.726} C_VEL
LIN {X 0,Y 474.634,Z 129.365,A -85,B 0,C 180,E1 -7167.788,E2 -7167.788} C_VEL
LIN {X 0,Y 474.623,Z 129.359,A -85,B 0,C 180,E1 -7170.884,E2 -7170.884} C_VEL
LIN {X 0,Y 474.652,Z 129.362,A -85,B 0,C 180,E1 -7173.628,E2 -7173.628} C_VEL
LIN {X 0,Y 474.632,Z 129.358,A -85,B 0,C 180,E1 -7176.642,E2 -7176.642} C_VEL
LIN {X 0,Y 474.653,Z 129.358,A -85,B 0,C 180,E1 -7180.09,E2 -7180.09} C_VEL
LIN {X 0,Y 474.649,Z 129.357,A -85,B 0,C 180,E1 -7182.775,E2 -7182.775} C_VEL
LIN {X 0,Y 474.65,Z 129.364,A -85,B 0,C 180,E1 -7185.421,E2 -7185.421} C_VEL
LIN {X 0,Y 474.702,Z 129.351,A -85,B 0,C 180,E1 -7188.038,E2 -7188.038} C_VEL
LIN {X 0,Y 474.727,Z 129.352,A -85,B 0,C 180,E1 -7191.487,E2 -7191.487} C_VEL
LIN {X 0,Y 474.78,Z 129.34,A -85,B 0,C 180,E1 -7194.053,E2 -7194.053} C_VEL
LIN {X 0,Y 474.893,Z 129.33,A -85,B 0,C 180,E1 -7197.456,E2 -7197.456} C_VEL
LIN {X 0,Y 474.911,Z 129.324,A -85,B 0,C 180,E1 -7200,E2 -7200} C_VEL
LIN {X 0,Y 474.893,Z 129.328,A -85,B 0,C 180,E1 -7202.545,E2 -7202.545} C_VEL
LIN {X 0,Y 474.769,Z 129.341,A -85,B 0,C 180,E1 -7205.948,E2 -7205.948} C_VEL
LIN {X 0,Y 474.726,Z 129.35,A -85,B 0,C 180,E1 -7208.514,E2 -7208.514} C_VEL
LIN {X 0,Y 474.703,Z 129.35,A -85,B 0,C 180,E1 -7211.963,E2 -7211.963} C_VEL
LIN {X 0,Y 474.699,Z 129.35,A -85,B 0,C 180,E1 -7215.456,E2 -7215.456} C_VEL
LIN {X 0,Y 474.665,Z 129.357,A -85,B 0,C 180,E1 -7219.01,E2 -7219.01} C_VEL
LIN {X 0,Y 474.587,Z 129.364,A -85,B 0,C 180,E1 -7221.729,E2 -7221.729} C_VEL
LIN {X 0,Y 474.656,Z 129.364,A -85,B 0,C 180,E1 -7224.493,E2 -7224.493} C_VEL
LIN {X 0,Y 474.68,Z 129.352,A -85,B 0,C 180,E1 -7227.335,E2 -7227.335} C_VEL
LIN {X 0,Y 474.605,Z 129.368,A -85,B 0,C 180,E1 -7230.23,E2 -7230.23} C_VEL
LIN {X 0,Y 474.642,Z 129.357,A -85,B 0,C 180,E1 -7233.22,E2 -7233.22} C_VEL
LIN {X 0,Y 474.589,Z 129.37,A -85,B 0,C 180,E1 -7236.324,E2 -7236.324} C_VEL
LIN {X 0,Y 474.651,Z 129.358,A -85,B 0,C 180,E1 -7239.651,E2 -7239.651} C_VEL
LIN {X 0,Y 474.616,Z 129.36,A -85,B 0,C 180,E1 -7242.934,E2 -7242.934} C_VEL
LIN {X 0,Y 474.61,Z 129.368,A -85,B 0,C 180,E1 -7245.896,E2 -7245.896} C_VEL
LIN {X 0,Y 474.642,Z 129.357,A -85,B 0,C 180,E1 -7249.039,E2 -7249.039} C_VEL
LIN {X 0,Y 474.617,Z 129.367,A -85,B 0,C 180,E1 -7251.703,E2 -7251.703} C_VEL
LIN {X 0,Y 474.626,Z 129.359,A -85,B 0,C 180,E1 -7254.726,E2 -7254.726} C_VEL
LIN {X 0,Y 474.637,Z 129.364,A -85,B 0,C 180,E1 -7257.788,E2 -7257.788} C_VEL
LIN {X 0,Y 474.626,Z 129.363,A -85,B 0,C 180,E1 -7260.885,E2 -7260.885} C_VEL
LIN {X 0,Y 474.767,Z 129.491,A -85,B 0,C 180,E1 -7263.309,E2 -7263.309} C_VEL
LIN {X 0,Y 476.968,Z 141.304,A -85,B 0,C 180,E1 -7265.402,E2 -7265.402} C_VEL
LIN {X 0,Y 476.39,Z 156.569,A -85,B 0,C 180,E1 -7267.902,E2 -7267.902} C_VEL
LIN {X 0,Y 475.658,Z 178.715,A -85,B 0,C 180,E1 -7271.478,E2 -7271.478} C_VEL
LIN {X 0,Y 475.22,Z 189.767,A -85,B 0,C 180,E1 -7273.24,E2 -7273.24} C_VEL
LIN {X 0,Y 477.917,Z 209.662,A -85,B 0,C 180,E1 -7273.655,E2 -7273.655} C_VEL
LIN {X 0,Y 477.282,Z 298.471,A -85,B 0,C 180,E1 -7275.04,E2 -7275.04} C_VEL
LIN {X 0,Y 476.873,Z 311.731,A -85,B 0,C 180,E1 -7275.409,E2 -7275.409} C_VEL
LIN {X 0,Y 476.397,Z 325.046,A -85,B 0,C 180,E1 -7275.966,E2 -7275.966} C_VEL
LIN {X 0,Y 475.941,Z 337.039,A -85,B 0,C 180,E1 -7276.66,E2 -7276.66} C_VEL
LIN {X 0,Y 475.439,Z 349.266,A -85,B 0,C 180,E1 -7277.575,E2 -7277.575} C_VEL
LIN {X 0,Y 475.049,Z 358.922,A -85,B 0,C 180,E1 -7278.479,E2 -7278.479} C_VEL
LIN {X 0,Y 474.581,Z 368.238,A -85,B 0,C 180,E1 -7279.548,E2 -7279.548} C_VEL
LIN {X 0,Y 474.246,Z 377.292,A -85,B 0,C 180,E1 -7280.833,E2 -7280.833} C_VEL
LIN {X 0,Y 474.027,Z 384.586,A -85,B 0,C 180,E1 -7282.118,E2 -7282.118} C_VEL
LIN {X 0,Y 473.854,Z 391.086,A -85,B 0,C 180,E1 -7283.575,E2 -7283.575} C_VEL
LIN {X 0,Y 473.823,Z 395.628,A -85,B 0,C 180,E1 -7284.894,E2 -7284.894} C_VEL
LIN {X 0,Y 473.75,Z 397.946,A -85,B 0,C 180,E1 -7285.746,E2 -7285.746} C_VEL
LIN {X 0,Y 473.841,Z 399.836,A -85,B 0,C 180,E1 -7286.599,E2 -7286.599} C_VEL
LIN {X 0,Y 473.793,Z 401.247,A -85,B 0,C 180,E1 -7287.449,E2 -7287.449} C_VEL
LIN {X 0,Y 473.761,Z 402.248,A -85,B 0,C 180,E1 -7288.3,E2 -7288.3} C_VEL
LIN {X 0,Y 473.693,Z 403.065,A -85,B 0,C 180,E1 -7290,E2 -7290} C_VEL
LIN {X 0,Y 473.761,Z 402.217,A -85,B 0,C 180,E1 -7291.7,E2 -7291.7} C_VEL
LIN {X 0,Y 473.793,Z 401.199,A -85,B 0,C 180,E1 -7292.55,E2 -7292.55} C_VEL
LIN {X 0,Y 473.841,Z 399.776,A -85,B 0,C 180,E1 -7293.401,E2 -7293.401} C_VEL
LIN {X 0,Y 473.762,Z 396.78,A -85,B 0,C 180,E1 -7294.68,E2 -7294.68} C_VEL
LIN {X 0,Y 473.798,Z 392.736,A -85,B 0,C 180,E1 -7295.96,E2 -7295.96} C_VEL
LIN {X 0,Y 473.998,Z 386.529,A -85,B 0,C 180,E1 -7297.454,E2 -7297.454} C_VEL
LIN {X 0,Y 474.142,Z 379.751,A -85,B 0,C 180,E1 -7298.739,E2 -7298.739} C_VEL
LIN {X 0,Y 474.429,Z 371.353,A -85,B 0,C 180,E1 -7300.024,E2 -7300.024} C_VEL
LIN {X 0,Y 474.836,Z 362.741,A -85,B 0,C 180,E1 -7301.093,E2 -7301.093} C_VEL
LIN {X 0,Y 475.264,Z 352.649,A -85,B 0,C 180,E1 -7302.116,E2 -7302.116} C_VEL
LIN {X 0,Y 475.718,Z 341.601,A -85,B 0,C 180,E1 -7303.02,E2 -7303.02} C_VEL
LIN {X 0,Y 476.211,Z 330.064,A -85,B 0,C 180,E1 -7303.767,E2 -7303.767} C_VEL
LIN {X 0,Y 476.665,Z 318.138,A -85,B 0,C 180,E1 -7304.352,E2 -7304.352} C_VEL
LIN {X 0,Y 477.119,Z 305.329,A -85,B 0,C 180,E1 -7304.802,E2 -7304.802} C_VEL
LIN {X 0,Y 477.404,Z 292.094,A -85,B 0,C 180,E1 -7305.093,E2 -7305.093} C_VEL
LIN {X 0,Y 477.883,Z 208.54,A -85,B 0,C 180,E1 -7306.388,E2 -7306.388} C_VEL
LIN {X 0,Y 475.242,Z 188.959,A -85,B 0,C 180,E1 -7306.808,E2 -7306.808} C_VEL
LIN {X 0,Y 475.814,Z 168.327,A -85,B 0,C 180,E1 -7310.085,E2 -7310.085} C_VEL
LIN {X 0,Y 476.51,Z 150.131,A -85,B 0,C 180,E1 -7313.007,E2 -7313.007} C_VEL
LIN {X 0,Y 476.755,Z 140.29,A -85,B 0,C 180,E1 -7314.61,E2 -7314.61} C_VEL
LIN {X 0,Y 474.709,Z 129.357,A -85,B 0,C 180,E1 -7316.546,E2 -7316.546} C_VEL
LIN {X 0,Y 474.623,Z 129.365,A -85,B 0,C 180,E1 -7319.252,E2 -7319.252} C_VEL
LIN {X 0,Y 474.616,Z 129.368,A -85,B 0,C 180,E1 -7322.43,E2 -7322.43} C_VEL
LIN {X 0,Y 474.615,Z 129.363,A -85,B 0,C 180,E1 -7325.469,E2 -7325.469} C_VEL
LIN {X 0,Y 474.623,Z 129.367,A -85,B 0,C 180,E1 -7328.456,E2 -7328.456} C_VEL
LIN {X 0,Y 474.642,Z 129.36,A -85,B 0,C 180,E1 -7330.961,E2 -7330.961} C_VEL
LIN {X 0,Y 474.61,Z 129.37,A -85,B 0,C 180,E1 -7334.104,E2 -7334.104} C_VEL
LIN {X 0,Y 474.615,Z 129.363,A -85,B 0,C 180,E1 -7337.065,E2 -7337.065} C_VEL
LIN {X 0,Y 474.669,Z 129.355,A -85,B 0,C 180,E1 -7340.456,E2 -7340.456} C_VEL
LIN {X 0,Y 474.588,Z 129.37,A -85,B 0,C 180,E1 -7343.676,E2 -7343.676} C_VEL
LIN {X 0,Y 474.642,Z 129.356,A -85,B 0,C 180,E1 -7346.78,E2 -7346.78} C_VEL
LIN {X 0,Y 474.604,Z 129.367,A -85,B 0,C 180,E1 -7349.77,E2 -7349.77} C_VEL
LIN {X 0,Y 474.696,Z 129.35,A -85,B 0,C 180,E1 -7352.68,E2 -7352.68} C_VEL
LIN {X 0,Y 474.639,Z 129.363,A -85,B 0,C 180,E1 -7355.506,E2 -7355.506} C_VEL
LIN {X 0,Y 474.669,Z 129.356,A -85,B 0,C 180,E1 -7359.185,E2 -7359.185} C_VEL
LIN {X 0,Y 474.656,Z 129.358,A -85,B 0,C 180,E1 -7361.884,E2 -7361.884} C_VEL
LIN {X 0,Y 474.699,Z 129.348,A -85,B 0,C 180,E1 -7364.544,E2 -7364.544} C_VEL
LIN {X 0,Y 474.702,Z 129.348,A -85,B 0,C 180,E1 -7368.037,E2 -7368.037} C_VEL
LIN {X 0,Y 474.727,Z 129.35,A -85,B 0,C 180,E1 -7371.486,E2 -7371.486} C_VEL
LIN {X 0,Y 474.779,Z 129.341,A -85,B 0,C 180,E1 -7374.052,E2 -7374.052} C_VEL
LIN {X 0,Y 474.892,Z 129.33,A -85,B 0,C 180,E1 -7377.455,E2 -7377.455} C_VEL
LIN {X 0,Y 474.91,Z 129.322,A -85,B 0,C 180,E1 -7380,E2 -7380} C_VEL
LIN {X 0,Y 474.893,Z 129.329,A -85,B 0,C 180,E1 -7382.544,E2 -7382.544} C_VEL
LIN {X 0,Y 474.769,Z 129.34,A -85,B 0,C 180,E1 -7385.948,E2 -7385.948} C_VEL
LIN {X 0,Y 474.726,Z 129.352,A -85,B 0,C 180,E1 -7388.513,E2 -7388.513} C_VEL
LIN {X 0,Y 474.702,Z 129.35,A -85,B 0,C 180,E1 -7391.962,E2 -7391.962} C_VEL
LIN {X 0,Y 474.697,Z 129.352,A -85,B 0,C 180,E1 -7395.456,E2 -7395.456} C_VEL
LIN {X 0,Y 474.663,Z 129.359,A -85,B 0,C 180,E1 -7399.01,E2 -7399.01} C_VEL
LIN {X 0,Y 474.586,Z 129.366,A -85,B 0,C 180,E1 -7401.729,E2 -7401.729} C_VEL
LIN {X 0,Y 474.655,Z 129.366,A -85,B 0,C 180,E1 -7404.493,E2 -7404.493} C_VEL
LIN {X 0,Y 474.697,Z 129.354,A -85,B 0,C 180,E1 -7407.339,E2 -7407.339} C_VEL
LIN {X 0,Y 474.603,Z 129.367,A -85,B 0,C 180,E1 -7410.81,E2 -7410.81} C_VEL
LIN {X 0,Y 474.691,Z 129.425,A -85,B 0,C 180,E1 -7413.78,E2 -7413.78} C_VEL
LIN {X 0,Y 475.667,Z 134.808,A -85,B 0,C 180,E1 -7414.927,E2 -7414.927} C_VEL
LIN {X 0,Y 475.677,Z 141.708,A -85,B 0,C 180,E1 -7416.293,E2 -7416.293} C_VEL
LIN {X 0,Y 478.296,Z 154.717,A -85,B 0,C 180,E1 -7416.601,E2 -7416.601} C_VEL
LIN {X 0,Y 477.498,Z 248.761,A -85,B 0,C 180,E1 -7418.083,E2 -7418.083} C_VEL
LIN {X 0,Y 477.21,Z 262.24,A -85,B 0,C 180,E1 -7418.475,E2 -7418.475} C_VEL
LIN {X 0,Y 476.965,Z 273.473,A -85,B 0,C 180,E1 -7418.955,E2 -7418.955} C_VEL
LIN {X 0,Y 476.611,Z 285.248,A -85,B 0,C 180,E1 -7419.624,E2 -7419.624} C_VEL
LIN {X 0,Y 476.179,Z 297.008,A -85,B 0,C 180,E1 -7420.496,E2 -7420.496} C_VEL
LIN {X 0,Y 475.67,Z 308.007,A -85,B 0,C 180,E1 -7421.523,E2 -7421.523} C_VEL
LIN {X 0,Y 475.227,Z 316.989,A -85,B 0,C 180,E1 -7422.566,E2 -7422.566} C_VEL
LIN {X 0,Y 474.785,Z 325.867,A -85,B 0,C 180,E1 -7423.841,E2 -7423.841} C_VEL
LIN {X 0,Y 474.471,Z 332.634,A -85,B 0,C 180,E1 -7425.042,E2 -7425.042} C_VEL
LIN {X 0,Y 474.249,Z 338.147,A -85,B 0,C 180,E1 -7426.25,E2 -7426.25} C_VEL
LIN {X 0,Y 474.07,Z 342.567,A -85,B 0,C 180,E1 -7427.461,E2 -7427.461} C_VEL
LIN {X 0,Y 473.941,Z 346.021,A -85,B 0,C 180,E1 -7428.68,E2 -7428.68} C_VEL
LIN {X 0,Y 473.783,Z 349.333,A -85,B 0,C 180,E1 -7430.368,E2 -7430.368} C_VEL
LIN {X 0,Y 473.691,Z 350.898,A -85,B 0,C 180,E1 -7431.929,E2 -7431.929} C_VEL
LIN {X 0,Y 472.997,Z 351.238,A -85,B 0,C 180,E1 -7432.639,E2 -7432.639} C_VEL
LIN {X 0,Y 470.117,Z 351.273,A -85,B 0,C 180,E1 -7433.792,E2 -7433.792} C_VEL
LIN {X 0,Y 467.729,Z 350.764,A -85,B 0,C 180,E1 -7434.72,E2 -7434.72} C_VEL
LIN {X 0,Y 466.747,Z 350.034,A -85,B 0,C 180,E1 -7435.432,E2 -7435.432} C_VEL
LIN {X 0,Y 466.69,Z 349.689,A -85,B 0,C 180,E1 -7435.672,E2 -7435.672} C_VEL
LIN {X 0,Y 466.832,Z 346.936,A -85,B 0,C 180,E1 -7437.183,E2 -7437.183} C_VEL
LIN {X 0,Y 467.002,Z 342.829,A -85,B 0,C 180,E1 -7438.675,E2 -7438.675} C_VEL
LIN {X 0,Y 467.272,Z 336.965,A -85,B 0,C 180,E1 -7440.242,E2 -7440.242} C_VEL
LIN {X 0,Y 467.514,Z 330.97,A -85,B 0,C 180,E1 -7441.492,E2 -7441.492} C_VEL
LIN {X 0,Y 467.877,Z 323.587,A -85,B 0,C 180,E1 -7442.736,E2 -7442.736} C_VEL
LIN {X 0,Y 468.301,Z 314.361,A -85,B 0,C 180,E1 -7443.986,E2 -7443.986} C_VEL
LIN {X 0,Y 468.825,Z 304.53,A -85,B 0,C 180,E1 -7445.064,E2 -7445.064} C_VEL
LIN {X 0,Y 469.254,Z 293.851,A -85,B 0,C 180,E1 -7446.007,E2 -7446.007} C_VEL
LIN {X 0,Y 469.67,Z 283.215,A -85,B 0,C 180,E1 -7446.755,E2 -7446.755} C_VEL
LIN {X 0,Y 470.054,Z 270.58,A -85,B 0,C 180,E1 -7447.443,E2 -7447.443} C_VEL
LIN {X 0,Y 470.387,Z 258.184,A -85,B 0,C 180,E1 -7447.931,E2 -7447.931} C_VEL
LIN {X 0,Y 470.582,Z 245.739,A -85,B 0,C 180,E1 -7448.25,E2 -7448.25} C_VEL
LIN {X 0,Y 471.294,Z 154.749,A -85,B 0,C 180,E1 -7449.686,E2 -7449.686} C_VEL
LIN {X 0,Y 468.475,Z 141.193,A -85,B 0,C 180,E1 -7450.016,E2 -7450.016} C_VEL
LIN {X 0,Y 468.422,Z 135.262,A -85,B 0,C 180,E1 -7451.27,E2 -7451.27} C_VEL
LIN {X 0,Y 467.623,Z 130.238,A -85,B 0,C 180,E1 -7452.395,E2 -7452.395} C_VEL
LIN {X 0,Y 467.606,Z 130.238,A -85,B 0,C 180,E1 -7455.197,E2 -7455.197} C_VEL
LIN {X 0,Y 467.656,Z 130.233,A -85,B 0,C 180,E1 -7457.855,E2 -7457.855} C_VEL
LIN {X 0,Y 467.68,Z 130.23,A -85,B 0,C 180,E1 -7461.357,E2 -7461.357} C_VEL
LIN {X 0,Y 467.735,Z 130.22,A -85,B 0,C 180,E1 -7463.963,E2 -7463.963} C_VEL
LIN {X 0,Y 467.859,Z 130.21,A -85,B 0,C 180,E1 -7467.417,E2 -7467.417} C_VEL
LIN {X 0,Y 467.882,Z 130.2,A -85,B 0,C 180,E1 -7470,E2 -7470} C_VEL
LIN {X 0,Y 467.859,Z 130.203,A -85,B 0,C 180,E1 -7472.583,E2 -7472.583} C_VEL
LIN {X 0,Y 467.724,Z 130.219,A -85,B 0,C 180,E1 -7476.038,E2 -7476.038} C_VEL
LIN {X 0,Y 467.66,Z 130.23,A -85,B 0,C 180,E1 -7479.515,E2 -7479.515} C_VEL
LIN {X 0,Y 467.654,Z 130.228,A -85,B 0,C 180,E1 -7482.358,E2 -7482.358} C_VEL
LIN {X 0,Y 467.649,Z 130.228,A -85,B 0,C 180,E1 -7485.885,E2 -7485.885} C_VEL
LIN {X 0,Y 467.622,Z 130.234,A -85,B 0,C 180,E1 -7489.308,E2 -7489.308} C_VEL
LIN {X 0,Y 467.534,Z 130.243,A -85,B 0,C 180,E1 -7492.074,E2 -7492.074} C_VEL
